REGION Network 11: Е | Ж | З | И | Й |
   RUNG wire#powerrail
      I_Contact( #DONE )
      { S7_Templates := "SrcType := WChar" } EQ_Contact(in1 := #UNICODE, in2 := WCHAR#'Е')
      Move(in := 16#C5, out1 => #ASCII_HEX)
      S_Coil( #DONE )
   END_RUNG
   RUNG wire#powerrail
      I_Contact( #DONE )
      { S7_Templates := "SrcType := WChar" } EQ_Contact(in1 := #UNICODE, in2 := WCHAR#'Ж')
      Move(in := 16#C6, out1 => #ASCII_HEX)
      S_Coil( #DONE )
   END_RUNG
   RUNG wire#powerrail
      I_Contact( #DONE )
      { S7_Templates := "SrcType := WChar" } EQ_Contact(in1 := #UNICODE, in2 := WCHAR#'З')
      Move(in := 16#C7, out1 => #ASCII_HEX)
      S_Coil( #DONE )
   END_RUNG
   RUNG wire#powerrail
      I_Contact( #DONE )
      { S7_Templates := "SrcType := WChar" } EQ_Contact(in1 := #UNICODE, in2 := WCHAR#'И')
      Move(in := 16#C8, out1 => #ASCII_HEX)
      S_Coil( #DONE )
   END_RUNG
   RUNG wire#powerrail
      I_Contact( #DONE )
      { S7_Templates := "SrcType := WChar" } EQ_Contact(in1 := #UNICODE, in2 := WCHAR#'Й')
      Move(in := 16#C9, out1 => #ASCII_HEX)
      S_Coil( #DONE )
   END_RUNG
   // the same network as SCL:
   IF NOT #DONE AND (#UNICODE = WCHAR#'Е') THEN
       #ASCII_HEX := 16#C5;
       #DONE := TRUE;
   END_IF;
   IF NOT #DONE AND (#UNICODE = WCHAR#'Ж') THEN
       #ASCII_HEX := 16#C6;
       #DONE := TRUE;
   END_IF;
   IF NOT #DONE AND (#UNICODE = WCHAR#'З') THEN
       #ASCII_HEX := 16#C7;
       #DONE := TRUE;
   END_IF;
   IF NOT #DONE AND (#UNICODE = WCHAR#'И') THEN
       #ASCII_HEX := 16#C8;
       #DONE := TRUE;
   END_IF;
   IF NOT #DONE AND (#UNICODE = WCHAR#'Й') THEN
       #ASCII_HEX := 16#C9;
       #DONE := TRUE;
   END_IF;
END_REGION

REGION Network 12: К | Л | М | Н | О |
   RUNG wire#powerrail
      I_Contact( #DONE )
      { S7_Templates := "SrcType := WChar" } EQ_Contact(in1 := #UNICODE, in2 := WCHAR#'К')
      Move(in := 16#CA, out1 => #ASCII_HEX)
      S_Coil( #DONE )
   END_RUNG
   RUNG wire#powerrail
      I_Contact( #DONE )
      { S7_Templates := "SrcType := WChar" } EQ_Contact(in1 := #UNICODE, in2 := WCHAR#'Л')
      Move(in := 16#CB, out1 => #ASCII_HEX)
      S_Coil( #DONE )
   END_RUNG
   RUNG wire#powerrail
      I_Contact( #DONE )
      { S7_Templates := "SrcType := WChar" } EQ_Contact(in1 := #UNICODE, in2 := WCHAR#'М')
      Move(in := 16#CC, out1 => #ASCII_HEX)
      S_Coil( #DONE )
   END_RUNG
   RUNG wire#powerrail
      I_Contact( #DONE )
      { S7_Templates := "SrcType := WChar" } EQ_Contact(in1 := #UNICODE, in2 := WCHAR#'Н')
      Move(in := 16#CD, out1 => #ASCII_HEX)
      S_Coil( #DONE )
   END_RUNG
   RUNG wire#powerrail
      I_Contact( #DONE )
      { S7_Templates := "SrcType := WChar" } EQ_Contact(in1 := #UNICODE, in2 := WCHAR#'О')
      Move(in := 16#CE, out1 => #ASCII_HEX)
      S_Coil( #DONE )
   END_RUNG
   // the same network as SCL:
   IF NOT #DONE AND (#UNICODE = WCHAR#'К') THEN
       #ASCII_HEX := 16#CA;
       #DONE := TRUE;
   END_IF;
   IF NOT #DONE AND (#UNICODE = WCHAR#'Л') THEN
       #ASCII_HEX := 16#CB;
       #DONE := TRUE;
   END_IF;
   IF NOT #DONE AND (#UNICODE = WCHAR#'М') THEN
       #ASCII_HEX := 16#CC;
       #DONE := TRUE;
   END_IF;
   IF NOT #DONE AND (#UNICODE = WCHAR#'Н') THEN
       #ASCII_HEX := 16#CD;
       #DONE := TRUE;
   END_IF;
   IF NOT #DONE AND (#UNICODE = WCHAR#'О') THEN
       #ASCII_HEX := 16#CE;
       #DONE := TRUE;
   END_IF;
END_REGION

REGION Network 13: П | Р | С | Т | У |
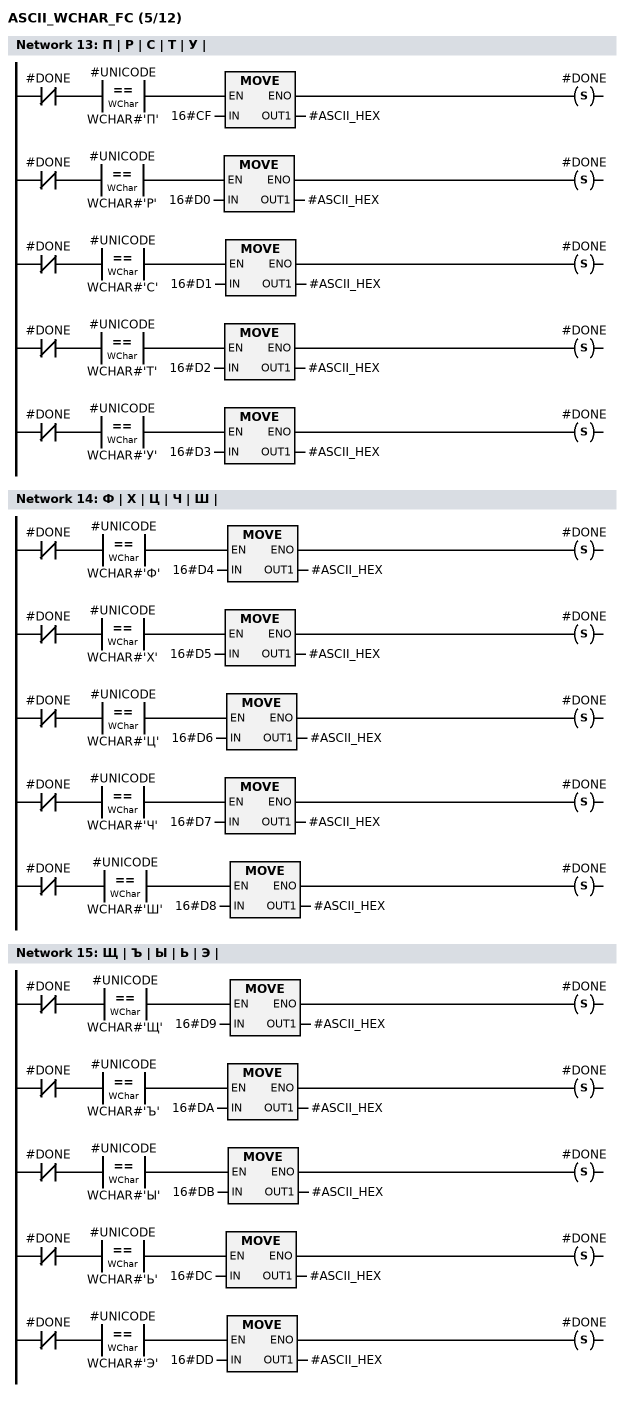
   RUNG wire#powerrail
      I_Contact( #DONE )
      { S7_Templates := "SrcType := WChar" } EQ_Contact(in1 := #UNICODE, in2 := WCHAR#'П')
      Move(in := 16#CF, out1 => #ASCII_HEX)
      S_Coil( #DONE )
   END_RUNG
   RUNG wire#powerrail
      I_Contact( #DONE )
      { S7_Templates := "SrcType := WChar" } EQ_Contact(in1 := #UNICODE, in2 := WCHAR#'Р')
      Move(in := 16#D0, out1 => #ASCII_HEX)
      S_Coil( #DONE )
   END_RUNG
   RUNG wire#powerrail
      I_Contact( #DONE )
      { S7_Templates := "SrcType := WChar" } EQ_Contact(in1 := #UNICODE, in2 := WCHAR#'С')
      Move(in := 16#D1, out1 => #ASCII_HEX)
      S_Coil( #DONE )
   END_RUNG
   RUNG wire#powerrail
      I_Contact( #DONE )
      { S7_Templates := "SrcType := WChar" } EQ_Contact(in1 := #UNICODE, in2 := WCHAR#'Т')
      Move(in := 16#D2, out1 => #ASCII_HEX)
      S_Coil( #DONE )
   END_RUNG
   RUNG wire#powerrail
      I_Contact( #DONE )
      { S7_Templates := "SrcType := WChar" } EQ_Contact(in1 := #UNICODE, in2 := WCHAR#'У')
      Move(in := 16#D3, out1 => #ASCII_HEX)
      S_Coil( #DONE )
   END_RUNG
   // the same network as SCL:
   IF NOT #DONE AND (#UNICODE = WCHAR#'П') THEN
       #ASCII_HEX := 16#CF;
       #DONE := TRUE;
   END_IF;
   IF NOT #DONE AND (#UNICODE = WCHAR#'Р') THEN
       #ASCII_HEX := 16#D0;
       #DONE := TRUE;
   END_IF;
   IF NOT #DONE AND (#UNICODE = WCHAR#'С') THEN
       #ASCII_HEX := 16#D1;
       #DONE := TRUE;
   END_IF;
   IF NOT #DONE AND (#UNICODE = WCHAR#'Т') THEN
       #ASCII_HEX := 16#D2;
       #DONE := TRUE;
   END_IF;
   IF NOT #DONE AND (#UNICODE = WCHAR#'У') THEN
       #ASCII_HEX := 16#D3;
       #DONE := TRUE;
   END_IF;
END_REGION

REGION Network 14: Ф | Х | Ц | Ч | Ш |
   RUNG wire#powerrail
      I_Contact( #DONE )
      { S7_Templates := "SrcType := WChar" } EQ_Contact(in1 := #UNICODE, in2 := WCHAR#'Ф')
      Move(in := 16#D4, out1 => #ASCII_HEX)
      S_Coil( #DONE )
   END_RUNG
   RUNG wire#powerrail
      I_Contact( #DONE )
      { S7_Templates := "SrcType := WChar" } EQ_Contact(in1 := #UNICODE, in2 := WCHAR#'Х')
      Move(in := 16#D5, out1 => #ASCII_HEX)
      S_Coil( #DONE )
   END_RUNG
   RUNG wire#powerrail
      I_Contact( #DONE )
      { S7_Templates := "SrcType := WChar" } EQ_Contact(in1 := #UNICODE, in2 := WCHAR#'Ц')
      Move(in := 16#D6, out1 => #ASCII_HEX)
      S_Coil( #DONE )
   END_RUNG
   RUNG wire#powerrail
      I_Contact( #DONE )
      { S7_Templates := "SrcType := WChar" } EQ_Contact(in1 := #UNICODE, in2 := WCHAR#'Ч')
      Move(in := 16#D7, out1 => #ASCII_HEX)
      S_Coil( #DONE )
   END_RUNG
   RUNG wire#powerrail
      I_Contact( #DONE )
      { S7_Templates := "SrcType := WChar" } EQ_Contact(in1 := #UNICODE, in2 := WCHAR#'Ш')
      Move(in := 16#D8, out1 => #ASCII_HEX)
      S_Coil( #DONE )
   END_RUNG
   // the same network as SCL:
   IF NOT #DONE AND (#UNICODE = WCHAR#'Ф') THEN
       #ASCII_HEX := 16#D4;
       #DONE := TRUE;
   END_IF;
   IF NOT #DONE AND (#UNICODE = WCHAR#'Х') THEN
       #ASCII_HEX := 16#D5;
       #DONE := TRUE;
   END_IF;
   IF NOT #DONE AND (#UNICODE = WCHAR#'Ц') THEN
       #ASCII_HEX := 16#D6;
       #DONE := TRUE;
   END_IF;
   IF NOT #DONE AND (#UNICODE = WCHAR#'Ч') THEN
       #ASCII_HEX := 16#D7;
       #DONE := TRUE;
   END_IF;
   IF NOT #DONE AND (#UNICODE = WCHAR#'Ш') THEN
       #ASCII_HEX := 16#D8;
       #DONE := TRUE;
   END_IF;
END_REGION

REGION Network 15: Щ | Ъ | Ы | Ь | Э |
   RUNG wire#powerrail
      I_Contact( #DONE )
      { S7_Templates := "SrcType := WChar" } EQ_Contact(in1 := #UNICODE, in2 := WCHAR#'Щ')
      Move(in := 16#D9, out1 => #ASCII_HEX)
      S_Coil( #DONE )
   END_RUNG
   RUNG wire#powerrail
      I_Contact( #DONE )
      { S7_Templates := "SrcType := WChar" } EQ_Contact(in1 := #UNICODE, in2 := WCHAR#'Ъ')
      Move(in := 16#DA, out1 => #ASCII_HEX)
      S_Coil( #DONE )
   END_RUNG
   RUNG wire#powerrail
      I_Contact( #DONE )
      { S7_Templates := "SrcType := WChar" } EQ_Contact(in1 := #UNICODE, in2 := WCHAR#'Ы')
      Move(in := 16#DB, out1 => #ASCII_HEX)
      S_Coil( #DONE )
   END_RUNG
   RUNG wire#powerrail
      I_Contact( #DONE )
      { S7_Templates := "SrcType := WChar" } EQ_Contact(in1 := #UNICODE, in2 := WCHAR#'Ь')
      Move(in := 16#DC, out1 => #ASCII_HEX)
      S_Coil( #DONE )
   END_RUNG
   RUNG wire#powerrail
      I_Contact( #DONE )
      { S7_Templates := "SrcType := WChar" } EQ_Contact(in1 := #UNICODE, in2 := WCHAR#'Э')
      Move(in := 16#DD, out1 => #ASCII_HEX)
      S_Coil( #DONE )
   END_RUNG
   // the same network as SCL:
   IF NOT #DONE AND (#UNICODE = WCHAR#'Щ') THEN
       #ASCII_HEX := 16#D9;
       #DONE := TRUE;
   END_IF;
   IF NOT #DONE AND (#UNICODE = WCHAR#'Ъ') THEN
       #ASCII_HEX := 16#DA;
       #DONE := TRUE;
   END_IF;
   IF NOT #DONE AND (#UNICODE = WCHAR#'Ы') THEN
       #ASCII_HEX := 16#DB;
       #DONE := TRUE;
   END_IF;
   IF NOT #DONE AND (#UNICODE = WCHAR#'Ь') THEN
       #ASCII_HEX := 16#DC;
       #DONE := TRUE;
   END_IF;
   IF NOT #DONE AND (#UNICODE = WCHAR#'Э') THEN
       #ASCII_HEX := 16#DD;
       #DONE := TRUE;
   END_IF;
END_REGION

REGION Network 16: Ю | Я |
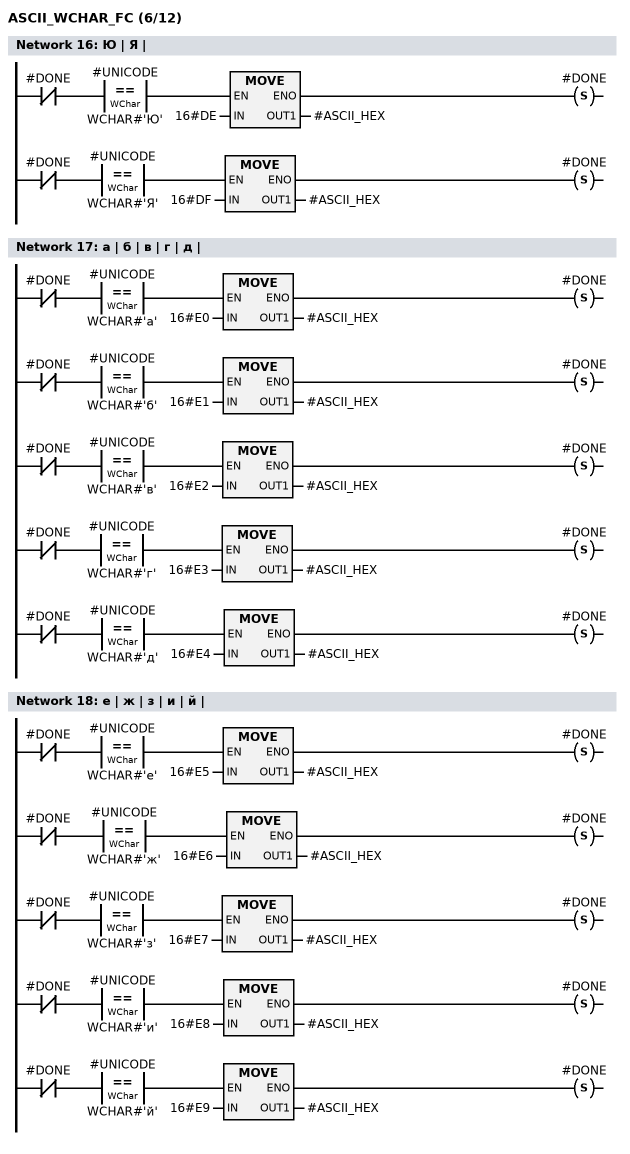
   RUNG wire#powerrail
      I_Contact( #DONE )
      { S7_Templates := "SrcType := WChar" } EQ_Contact(in1 := #UNICODE, in2 := WCHAR#'Ю')
      Move(in := 16#DE, out1 => #ASCII_HEX)
      S_Coil( #DONE )
   END_RUNG
   RUNG wire#powerrail
      I_Contact( #DONE )
      { S7_Templates := "SrcType := WChar" } EQ_Contact(in1 := #UNICODE, in2 := WCHAR#'Я')
      Move(in := 16#DF, out1 => #ASCII_HEX)
      S_Coil( #DONE )
   END_RUNG
   // the same network as SCL:
   IF NOT #DONE AND (#UNICODE = WCHAR#'Ю') THEN
       #ASCII_HEX := 16#DE;
       #DONE := TRUE;
   END_IF;
   IF NOT #DONE AND (#UNICODE = WCHAR#'Я') THEN
       #ASCII_HEX := 16#DF;
       #DONE := TRUE;
   END_IF;
END_REGION

REGION Network 17: а | б | в | г | д |
   RUNG wire#powerrail
      I_Contact( #DONE )
      { S7_Templates := "SrcType := WChar" } EQ_Contact(in1 := #UNICODE, in2 := WCHAR#'а')
      Move(in := 16#E0, out1 => #ASCII_HEX)
      S_Coil( #DONE )
   END_RUNG
   RUNG wire#powerrail
      I_Contact( #DONE )
      { S7_Templates := "SrcType := WChar" } EQ_Contact(in1 := #UNICODE, in2 := WCHAR#'б')
      Move(in := 16#E1, out1 => #ASCII_HEX)
      S_Coil( #DONE )
   END_RUNG
   RUNG wire#powerrail
      I_Contact( #DONE )
      { S7_Templates := "SrcType := WChar" } EQ_Contact(in1 := #UNICODE, in2 := WCHAR#'в')
      Move(in := 16#E2, out1 => #ASCII_HEX)
      S_Coil( #DONE )
   END_RUNG
   RUNG wire#powerrail
      I_Contact( #DONE )
      { S7_Templates := "SrcType := WChar" } EQ_Contact(in1 := #UNICODE, in2 := WCHAR#'г')
      Move(in := 16#E3, out1 => #ASCII_HEX)
      S_Coil( #DONE )
   END_RUNG
   RUNG wire#powerrail
      I_Contact( #DONE )
      { S7_Templates := "SrcType := WChar" } EQ_Contact(in1 := #UNICODE, in2 := WCHAR#'д')
      Move(in := 16#E4, out1 => #ASCII_HEX)
      S_Coil( #DONE )
   END_RUNG
   // the same network as SCL:
   IF NOT #DONE AND (#UNICODE = WCHAR#'а') THEN
       #ASCII_HEX := 16#E0;
       #DONE := TRUE;
   END_IF;
   IF NOT #DONE AND (#UNICODE = WCHAR#'б') THEN
       #ASCII_HEX := 16#E1;
       #DONE := TRUE;
   END_IF;
   IF NOT #DONE AND (#UNICODE = WCHAR#'в') THEN
       #ASCII_HEX := 16#E2;
       #DONE := TRUE;
   END_IF;
   IF NOT #DONE AND (#UNICODE = WCHAR#'г') THEN
       #ASCII_HEX := 16#E3;
       #DONE := TRUE;
   END_IF;
   IF NOT #DONE AND (#UNICODE = WCHAR#'д') THEN
       #ASCII_HEX := 16#E4;
       #DONE := TRUE;
   END_IF;
END_REGION

REGION Network 18: е | ж | з | и | й |
   RUNG wire#powerrail
      I_Contact( #DONE )
      { S7_Templates := "SrcType := WChar" } EQ_Contact(in1 := #UNICODE, in2 := WCHAR#'е')
      Move(in := 16#E5, out1 => #ASCII_HEX)
      S_Coil( #DONE )
   END_RUNG
   RUNG wire#powerrail
      I_Contact( #DONE )
      { S7_Templates := "SrcType := WChar" } EQ_Contact(in1 := #UNICODE, in2 := WCHAR#'ж')
      Move(in := 16#E6, out1 => #ASCII_HEX)
      S_Coil( #DONE )
   END_RUNG
   RUNG wire#powerrail
      I_Contact( #DONE )
      { S7_Templates := "SrcType := WChar" } EQ_Contact(in1 := #UNICODE, in2 := WCHAR#'з')
      Move(in := 16#E7, out1 => #ASCII_HEX)
      S_Coil( #DONE )
   END_RUNG
   RUNG wire#powerrail
      I_Contact( #DONE )
      { S7_Templates := "SrcType := WChar" } EQ_Contact(in1 := #UNICODE, in2 := WCHAR#'и')
      Move(in := 16#E8, out1 => #ASCII_HEX)
      S_Coil( #DONE )
   END_RUNG
   RUNG wire#powerrail
      I_Contact( #DONE )
      { S7_Templates := "SrcType := WChar" } EQ_Contact(in1 := #UNICODE, in2 := WCHAR#'й')
      Move(in := 16#E9, out1 => #ASCII_HEX)
      S_Coil( #DONE )
   END_RUNG
   // the same network as SCL:
   IF NOT #DONE AND (#UNICODE = WCHAR#'е') THEN
       #ASCII_HEX := 16#E5;
       #DONE := TRUE;
   END_IF;
   IF NOT #DONE AND (#UNICODE = WCHAR#'ж') THEN
       #ASCII_HEX := 16#E6;
       #DONE := TRUE;
   END_IF;
   IF NOT #DONE AND (#UNICODE = WCHAR#'з') THEN
       #ASCII_HEX := 16#E7;
       #DONE := TRUE;
   END_IF;
   IF NOT #DONE AND (#UNICODE = WCHAR#'и') THEN
       #ASCII_HEX := 16#E8;
       #DONE := TRUE;
   END_IF;
   IF NOT #DONE AND (#UNICODE = WCHAR#'й') THEN
       #ASCII_HEX := 16#E9;
       #DONE := TRUE;
   END_IF;
END_REGION

REGION Network 19: к | л | м | н | о |
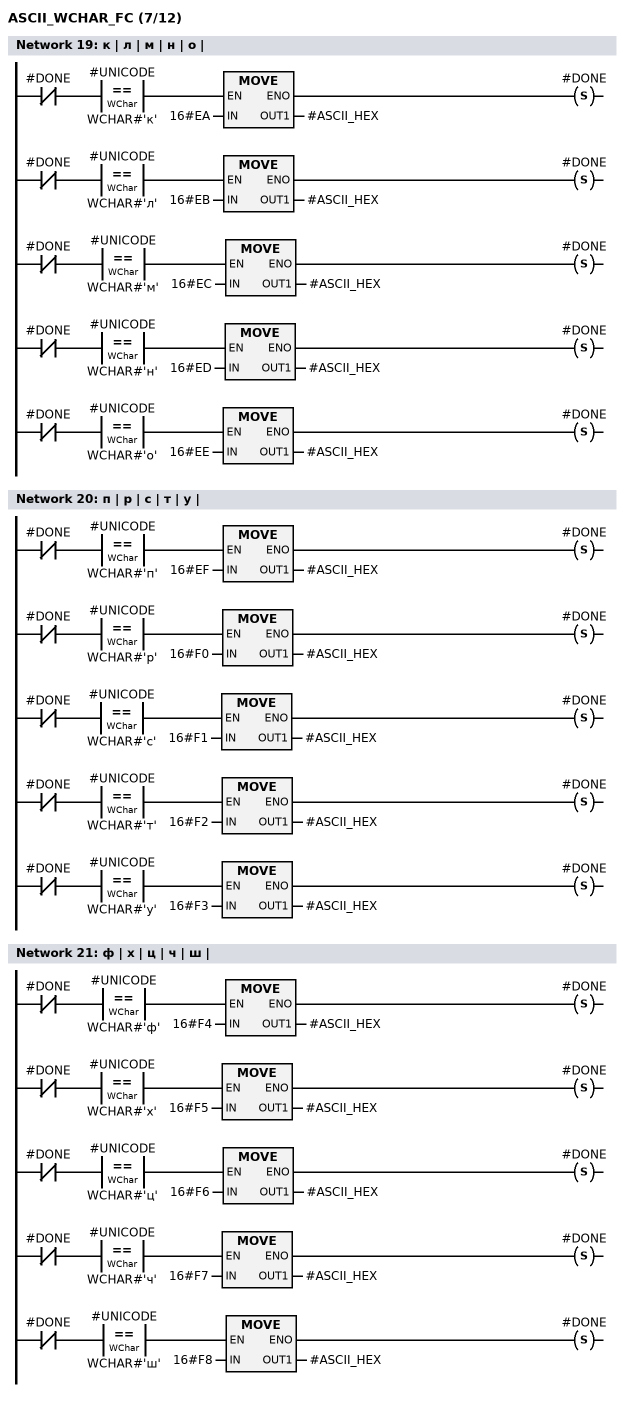
   RUNG wire#powerrail
      I_Contact( #DONE )
      { S7_Templates := "SrcType := WChar" } EQ_Contact(in1 := #UNICODE, in2 := WCHAR#'к')
      Move(in := 16#EA, out1 => #ASCII_HEX)
      S_Coil( #DONE )
   END_RUNG
   RUNG wire#powerrail
      I_Contact( #DONE )
      { S7_Templates := "SrcType := WChar" } EQ_Contact(in1 := #UNICODE, in2 := WCHAR#'л')
      Move(in := 16#EB, out1 => #ASCII_HEX)
      S_Coil( #DONE )
   END_RUNG
   RUNG wire#powerrail
      I_Contact( #DONE )
      { S7_Templates := "SrcType := WChar" } EQ_Contact(in1 := #UNICODE, in2 := WCHAR#'м')
      Move(in := 16#EC, out1 => #ASCII_HEX)
      S_Coil( #DONE )
   END_RUNG
   RUNG wire#powerrail
      I_Contact( #DONE )
      { S7_Templates := "SrcType := WChar" } EQ_Contact(in1 := #UNICODE, in2 := WCHAR#'н')
      Move(in := 16#ED, out1 => #ASCII_HEX)
      S_Coil( #DONE )
   END_RUNG
   RUNG wire#powerrail
      I_Contact( #DONE )
      { S7_Templates := "SrcType := WChar" } EQ_Contact(in1 := #UNICODE, in2 := WCHAR#'о')
      Move(in := 16#EE, out1 => #ASCII_HEX)
      S_Coil( #DONE )
   END_RUNG
   // the same network as SCL:
   IF NOT #DONE AND (#UNICODE = WCHAR#'к') THEN
       #ASCII_HEX := 16#EA;
       #DONE := TRUE;
   END_IF;
   IF NOT #DONE AND (#UNICODE = WCHAR#'л') THEN
       #ASCII_HEX := 16#EB;
       #DONE := TRUE;
   END_IF;
   IF NOT #DONE AND (#UNICODE = WCHAR#'м') THEN
       #ASCII_HEX := 16#EC;
       #DONE := TRUE;
   END_IF;
   IF NOT #DONE AND (#UNICODE = WCHAR#'н') THEN
       #ASCII_HEX := 16#ED;
       #DONE := TRUE;
   END_IF;
   IF NOT #DONE AND (#UNICODE = WCHAR#'о') THEN
       #ASCII_HEX := 16#EE;
       #DONE := TRUE;
   END_IF;
END_REGION

REGION Network 20: п | р | с | т | у |
   RUNG wire#powerrail
      I_Contact( #DONE )
      { S7_Templates := "SrcType := WChar" } EQ_Contact(in1 := #UNICODE, in2 := WCHAR#'п')
      Move(in := 16#EF, out1 => #ASCII_HEX)
      S_Coil( #DONE )
   END_RUNG
   RUNG wire#powerrail
      I_Contact( #DONE )
      { S7_Templates := "SrcType := WChar" } EQ_Contact(in1 := #UNICODE, in2 := WCHAR#'р')
      Move(in := 16#F0, out1 => #ASCII_HEX)
      S_Coil( #DONE )
   END_RUNG
   RUNG wire#powerrail
      I_Contact( #DONE )
      { S7_Templates := "SrcType := WChar" } EQ_Contact(in1 := #UNICODE, in2 := WCHAR#'с')
      Move(in := 16#F1, out1 => #ASCII_HEX)
      S_Coil( #DONE )
   END_RUNG
   RUNG wire#powerrail
      I_Contact( #DONE )
      { S7_Templates := "SrcType := WChar" } EQ_Contact(in1 := #UNICODE, in2 := WCHAR#'т')
      Move(in := 16#F2, out1 => #ASCII_HEX)
      S_Coil( #DONE )
   END_RUNG
   RUNG wire#powerrail
      I_Contact( #DONE )
      { S7_Templates := "SrcType := WChar" } EQ_Contact(in1 := #UNICODE, in2 := WCHAR#'у')
      Move(in := 16#F3, out1 => #ASCII_HEX)
      S_Coil( #DONE )
   END_RUNG
   // the same network as SCL:
   IF NOT #DONE AND (#UNICODE = WCHAR#'п') THEN
       #ASCII_HEX := 16#EF;
       #DONE := TRUE;
   END_IF;
   IF NOT #DONE AND (#UNICODE = WCHAR#'р') THEN
       #ASCII_HEX := 16#F0;
       #DONE := TRUE;
   END_IF;
   IF NOT #DONE AND (#UNICODE = WCHAR#'с') THEN
       #ASCII_HEX := 16#F1;
       #DONE := TRUE;
   END_IF;
   IF NOT #DONE AND (#UNICODE = WCHAR#'т') THEN
       #ASCII_HEX := 16#F2;
       #DONE := TRUE;
   END_IF;
   IF NOT #DONE AND (#UNICODE = WCHAR#'у') THEN
       #ASCII_HEX := 16#F3;
       #DONE := TRUE;
   END_IF;
END_REGION

REGION Network 21: ф | х | ц | ч | ш |
   RUNG wire#powerrail
      I_Contact( #DONE )
      { S7_Templates := "SrcType := WChar" } EQ_Contact(in1 := #UNICODE, in2 := WCHAR#'ф')
      Move(in := 16#F4, out1 => #ASCII_HEX)
      S_Coil( #DONE )
   END_RUNG
   RUNG wire#powerrail
      I_Contact( #DONE )
      { S7_Templates := "SrcType := WChar" } EQ_Contact(in1 := #UNICODE, in2 := WCHAR#'х')
      Move(in := 16#F5, out1 => #ASCII_HEX)
      S_Coil( #DONE )
   END_RUNG
   RUNG wire#powerrail
      I_Contact( #DONE )
      { S7_Templates := "SrcType := WChar" } EQ_Contact(in1 := #UNICODE, in2 := WCHAR#'ц')
      Move(in := 16#F6, out1 => #ASCII_HEX)
      S_Coil( #DONE )
   END_RUNG
   RUNG wire#powerrail
      I_Contact( #DONE )
      { S7_Templates := "SrcType := WChar" } EQ_Contact(in1 := #UNICODE, in2 := WCHAR#'ч')
      Move(in := 16#F7, out1 => #ASCII_HEX)
      S_Coil( #DONE )
   END_RUNG
   RUNG wire#powerrail
      I_Contact( #DONE )
      { S7_Templates := "SrcType := WChar" } EQ_Contact(in1 := #UNICODE, in2 := WCHAR#'ш')
      Move(in := 16#F8, out1 => #ASCII_HEX)
      S_Coil( #DONE )
   END_RUNG
   // the same network as SCL:
   IF NOT #DONE AND (#UNICODE = WCHAR#'ф') THEN
       #ASCII_HEX := 16#F4;
       #DONE := TRUE;
   END_IF;
   IF NOT #DONE AND (#UNICODE = WCHAR#'х') THEN
       #ASCII_HEX := 16#F5;
       #DONE := TRUE;
   END_IF;
   IF NOT #DONE AND (#UNICODE = WCHAR#'ц') THEN
       #ASCII_HEX := 16#F6;
       #DONE := TRUE;
   END_IF;
   IF NOT #DONE AND (#UNICODE = WCHAR#'ч') THEN
       #ASCII_HEX := 16#F7;
       #DONE := TRUE;
   END_IF;
   IF NOT #DONE AND (#UNICODE = WCHAR#'ш') THEN
       #ASCII_HEX := 16#F8;
       #DONE := TRUE;
   END_IF;
END_REGION

REGION Network 22: щ | ъ | ы | ь | э |
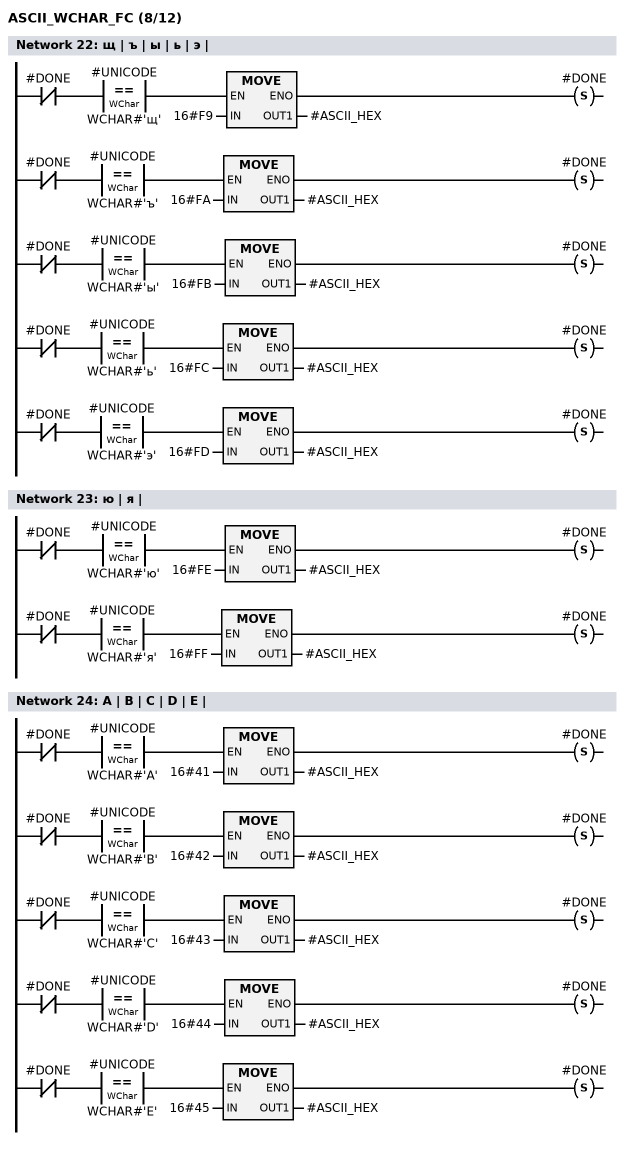
   RUNG wire#powerrail
      I_Contact( #DONE )
      { S7_Templates := "SrcType := WChar" } EQ_Contact(in1 := #UNICODE, in2 := WCHAR#'щ')
      Move(in := 16#F9, out1 => #ASCII_HEX)
      S_Coil( #DONE )
   END_RUNG
   RUNG wire#powerrail
      I_Contact( #DONE )
      { S7_Templates := "SrcType := WChar" } EQ_Contact(in1 := #UNICODE, in2 := WCHAR#'ъ')
      Move(in := 16#FA, out1 => #ASCII_HEX)
      S_Coil( #DONE )
   END_RUNG
   RUNG wire#powerrail
      I_Contact( #DONE )
      { S7_Templates := "SrcType := WChar" } EQ_Contact(in1 := #UNICODE, in2 := WCHAR#'ы')
      Move(in := 16#FB, out1 => #ASCII_HEX)
      S_Coil( #DONE )
   END_RUNG
   RUNG wire#powerrail
      I_Contact( #DONE )
      { S7_Templates := "SrcType := WChar" } EQ_Contact(in1 := #UNICODE, in2 := WCHAR#'ь')
      Move(in := 16#FC, out1 => #ASCII_HEX)
      S_Coil( #DONE )
   END_RUNG
   RUNG wire#powerrail
      I_Contact( #DONE )
      { S7_Templates := "SrcType := WChar" } EQ_Contact(in1 := #UNICODE, in2 := WCHAR#'э')
      Move(in := 16#FD, out1 => #ASCII_HEX)
      S_Coil( #DONE )
   END_RUNG
   // the same network as SCL:
   IF NOT #DONE AND (#UNICODE = WCHAR#'щ') THEN
       #ASCII_HEX := 16#F9;
       #DONE := TRUE;
   END_IF;
   IF NOT #DONE AND (#UNICODE = WCHAR#'ъ') THEN
       #ASCII_HEX := 16#FA;
       #DONE := TRUE;
   END_IF;
   IF NOT #DONE AND (#UNICODE = WCHAR#'ы') THEN
       #ASCII_HEX := 16#FB;
       #DONE := TRUE;
   END_IF;
   IF NOT #DONE AND (#UNICODE = WCHAR#'ь') THEN
       #ASCII_HEX := 16#FC;
       #DONE := TRUE;
   END_IF;
   IF NOT #DONE AND (#UNICODE = WCHAR#'э') THEN
       #ASCII_HEX := 16#FD;
       #DONE := TRUE;
   END_IF;
END_REGION

REGION Network 23: ю | я |
   RUNG wire#powerrail
      I_Contact( #DONE )
      { S7_Templates := "SrcType := WChar" } EQ_Contact(in1 := #UNICODE, in2 := WCHAR#'ю')
      Move(in := 16#FE, out1 => #ASCII_HEX)
      S_Coil( #DONE )
   END_RUNG
   RUNG wire#powerrail
      I_Contact( #DONE )
      { S7_Templates := "SrcType := WChar" } EQ_Contact(in1 := #UNICODE, in2 := WCHAR#'я')
      Move(in := 16#FF, out1 => #ASCII_HEX)
      S_Coil( #DONE )
   END_RUNG
   // the same network as SCL:
   IF NOT #DONE AND (#UNICODE = WCHAR#'ю') THEN
       #ASCII_HEX := 16#FE;
       #DONE := TRUE;
   END_IF;
   IF NOT #DONE AND (#UNICODE = WCHAR#'я') THEN
       #ASCII_HEX := 16#FF;
       #DONE := TRUE;
   END_IF;
END_REGION

REGION Network 24: A | B | C | D | E |
   RUNG wire#powerrail
      I_Contact( #DONE )
      { S7_Templates := "SrcType := WChar" } EQ_Contact(in1 := #UNICODE, in2 := WCHAR#'A')
      Move(in := 16#41, out1 => #ASCII_HEX)
      S_Coil( #DONE )
   END_RUNG
   RUNG wire#powerrail
      I_Contact( #DONE )
      { S7_Templates := "SrcType := WChar" } EQ_Contact(in1 := #UNICODE, in2 := WCHAR#'B')
      Move(in := 16#42, out1 => #ASCII_HEX)
      S_Coil( #DONE )
   END_RUNG
   RUNG wire#powerrail
      I_Contact( #DONE )
      { S7_Templates := "SrcType := WChar" } EQ_Contact(in1 := #UNICODE, in2 := WCHAR#'C')
      Move(in := 16#43, out1 => #ASCII_HEX)
      S_Coil( #DONE )
   END_RUNG
   RUNG wire#powerrail
      I_Contact( #DONE )
      { S7_Templates := "SrcType := WChar" } EQ_Contact(in1 := #UNICODE, in2 := WCHAR#'D')
      Move(in := 16#44, out1 => #ASCII_HEX)
      S_Coil( #DONE )
   END_RUNG
   RUNG wire#powerrail
      I_Contact( #DONE )
      { S7_Templates := "SrcType := WChar" } EQ_Contact(in1 := #UNICODE, in2 := WCHAR#'E')
      Move(in := 16#45, out1 => #ASCII_HEX)
      S_Coil( #DONE )
   END_RUNG
   // the same network as SCL:
   IF NOT #DONE AND (#UNICODE = WCHAR#'A') THEN
       #ASCII_HEX := 16#41;
       #DONE := TRUE;
   END_IF;
   IF NOT #DONE AND (#UNICODE = WCHAR#'B') THEN
       #ASCII_HEX := 16#42;
       #DONE := TRUE;
   END_IF;
   IF NOT #DONE AND (#UNICODE = WCHAR#'C') THEN
       #ASCII_HEX := 16#43;
       #DONE := TRUE;
   END_IF;
   IF NOT #DONE AND (#UNICODE = WCHAR#'D') THEN
       #ASCII_HEX := 16#44;
       #DONE := TRUE;
   END_IF;
   IF NOT #DONE AND (#UNICODE = WCHAR#'E') THEN
       #ASCII_HEX := 16#45;
       #DONE := TRUE;
   END_IF;
END_REGION

REGION Network 25: F | G | H | I | J |
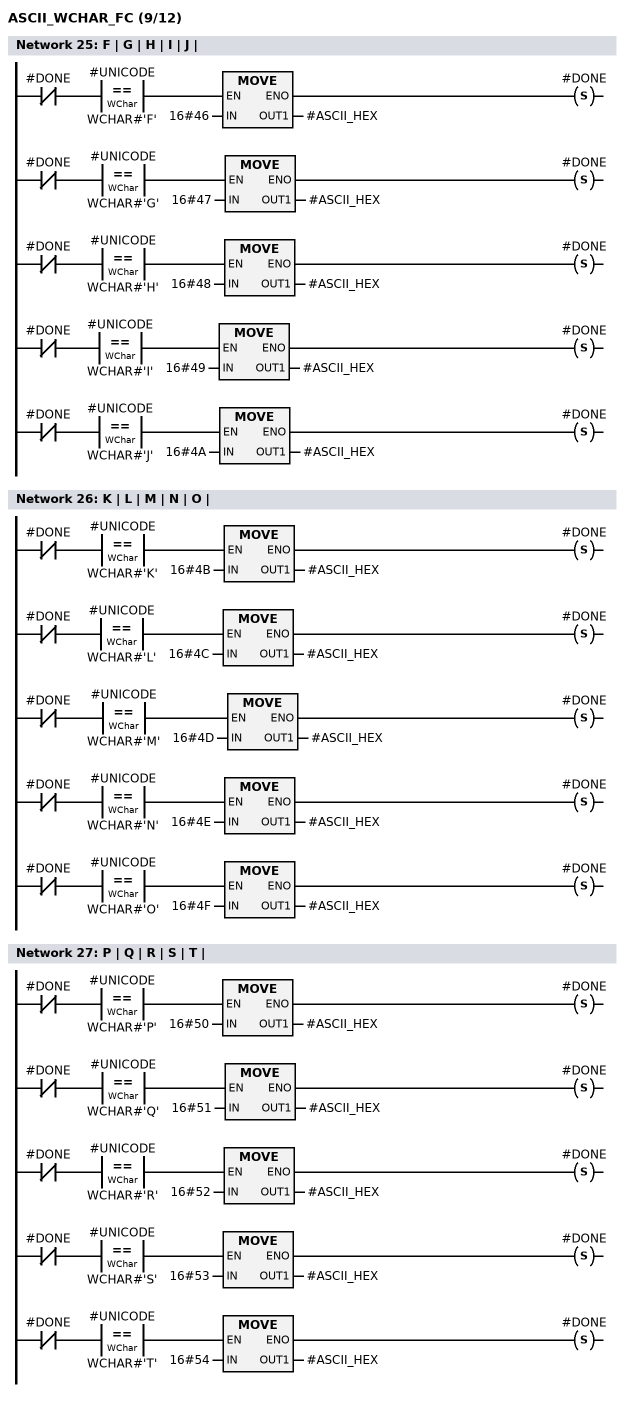
   RUNG wire#powerrail
      I_Contact( #DONE )
      { S7_Templates := "SrcType := WChar" } EQ_Contact(in1 := #UNICODE, in2 := WCHAR#'F')
      Move(in := 16#46, out1 => #ASCII_HEX)
      S_Coil( #DONE )
   END_RUNG
   RUNG wire#powerrail
      I_Contact( #DONE )
      { S7_Templates := "SrcType := WChar" } EQ_Contact(in1 := #UNICODE, in2 := WCHAR#'G')
      Move(in := 16#47, out1 => #ASCII_HEX)
      S_Coil( #DONE )
   END_RUNG
   RUNG wire#powerrail
      I_Contact( #DONE )
      { S7_Templates := "SrcType := WChar" } EQ_Contact(in1 := #UNICODE, in2 := WCHAR#'H')
      Move(in := 16#48, out1 => #ASCII_HEX)
      S_Coil( #DONE )
   END_RUNG
   RUNG wire#powerrail
      I_Contact( #DONE )
      { S7_Templates := "SrcType := WChar" } EQ_Contact(in1 := #UNICODE, in2 := WCHAR#'I')
      Move(in := 16#49, out1 => #ASCII_HEX)
      S_Coil( #DONE )
   END_RUNG
   RUNG wire#powerrail
      I_Contact( #DONE )
      { S7_Templates := "SrcType := WChar" } EQ_Contact(in1 := #UNICODE, in2 := WCHAR#'J')
      Move(in := 16#4A, out1 => #ASCII_HEX)
      S_Coil( #DONE )
   END_RUNG
   // the same network as SCL:
   IF NOT #DONE AND (#UNICODE = WCHAR#'F') THEN
       #ASCII_HEX := 16#46;
       #DONE := TRUE;
   END_IF;
   IF NOT #DONE AND (#UNICODE = WCHAR#'G') THEN
       #ASCII_HEX := 16#47;
       #DONE := TRUE;
   END_IF;
   IF NOT #DONE AND (#UNICODE = WCHAR#'H') THEN
       #ASCII_HEX := 16#48;
       #DONE := TRUE;
   END_IF;
   IF NOT #DONE AND (#UNICODE = WCHAR#'I') THEN
       #ASCII_HEX := 16#49;
       #DONE := TRUE;
   END_IF;
   IF NOT #DONE AND (#UNICODE = WCHAR#'J') THEN
       #ASCII_HEX := 16#4A;
       #DONE := TRUE;
   END_IF;
END_REGION

REGION Network 26: K | L | M | N | O |
   RUNG wire#powerrail
      I_Contact( #DONE )
      { S7_Templates := "SrcType := WChar" } EQ_Contact(in1 := #UNICODE, in2 := WCHAR#'K')
      Move(in := 16#4B, out1 => #ASCII_HEX)
      S_Coil( #DONE )
   END_RUNG
   RUNG wire#powerrail
      I_Contact( #DONE )
      { S7_Templates := "SrcType := WChar" } EQ_Contact(in1 := #UNICODE, in2 := WCHAR#'L')
      Move(in := 16#4C, out1 => #ASCII_HEX)
      S_Coil( #DONE )
   END_RUNG
   RUNG wire#powerrail
      I_Contact( #DONE )
      { S7_Templates := "SrcType := WChar" } EQ_Contact(in1 := #UNICODE, in2 := WCHAR#'M')
      Move(in := 16#4D, out1 => #ASCII_HEX)
      S_Coil( #DONE )
   END_RUNG
   RUNG wire#powerrail
      I_Contact( #DONE )
      { S7_Templates := "SrcType := WChar" } EQ_Contact(in1 := #UNICODE, in2 := WCHAR#'N')
      Move(in := 16#4E, out1 => #ASCII_HEX)
      S_Coil( #DONE )
   END_RUNG
   RUNG wire#powerrail
      I_Contact( #DONE )
      { S7_Templates := "SrcType := WChar" } EQ_Contact(in1 := #UNICODE, in2 := WCHAR#'O')
      Move(in := 16#4F, out1 => #ASCII_HEX)
      S_Coil( #DONE )
   END_RUNG
   // the same network as SCL:
   IF NOT #DONE AND (#UNICODE = WCHAR#'K') THEN
       #ASCII_HEX := 16#4B;
       #DONE := TRUE;
   END_IF;
   IF NOT #DONE AND (#UNICODE = WCHAR#'L') THEN
       #ASCII_HEX := 16#4C;
       #DONE := TRUE;
   END_IF;
   IF NOT #DONE AND (#UNICODE = WCHAR#'M') THEN
       #ASCII_HEX := 16#4D;
       #DONE := TRUE;
   END_IF;
   IF NOT #DONE AND (#UNICODE = WCHAR#'N') THEN
       #ASCII_HEX := 16#4E;
       #DONE := TRUE;
   END_IF;
   IF NOT #DONE AND (#UNICODE = WCHAR#'O') THEN
       #ASCII_HEX := 16#4F;
       #DONE := TRUE;
   END_IF;
END_REGION

REGION Network 27: P | Q | R | S | T |
   RUNG wire#powerrail
      I_Contact( #DONE )
      { S7_Templates := "SrcType := WChar" } EQ_Contact(in1 := #UNICODE, in2 := WCHAR#'P')
      Move(in := 16#50, out1 => #ASCII_HEX)
      S_Coil( #DONE )
   END_RUNG
   RUNG wire#powerrail
      I_Contact( #DONE )
      { S7_Templates := "SrcType := WChar" } EQ_Contact(in1 := #UNICODE, in2 := WCHAR#'Q')
      Move(in := 16#51, out1 => #ASCII_HEX)
      S_Coil( #DONE )
   END_RUNG
   RUNG wire#powerrail
      I_Contact( #DONE )
      { S7_Templates := "SrcType := WChar" } EQ_Contact(in1 := #UNICODE, in2 := WCHAR#'R')
      Move(in := 16#52, out1 => #ASCII_HEX)
      S_Coil( #DONE )
   END_RUNG
   RUNG wire#powerrail
      I_Contact( #DONE )
      { S7_Templates := "SrcType := WChar" } EQ_Contact(in1 := #UNICODE, in2 := WCHAR#'S')
      Move(in := 16#53, out1 => #ASCII_HEX)
      S_Coil( #DONE )
   END_RUNG
   RUNG wire#powerrail
      I_Contact( #DONE )
      { S7_Templates := "SrcType := WChar" } EQ_Contact(in1 := #UNICODE, in2 := WCHAR#'T')
      Move(in := 16#54, out1 => #ASCII_HEX)
      S_Coil( #DONE )
   END_RUNG
   // the same network as SCL:
   IF NOT #DONE AND (#UNICODE = WCHAR#'P') THEN
       #ASCII_HEX := 16#50;
       #DONE := TRUE;
   END_IF;
   IF NOT #DONE AND (#UNICODE = WCHAR#'Q') THEN
       #ASCII_HEX := 16#51;
       #DONE := TRUE;
   END_IF;
   IF NOT #DONE AND (#UNICODE = WCHAR#'R') THEN
       #ASCII_HEX := 16#52;
       #DONE := TRUE;
   END_IF;
   IF NOT #DONE AND (#UNICODE = WCHAR#'S') THEN
       #ASCII_HEX := 16#53;
       #DONE := TRUE;
   END_IF;
   IF NOT #DONE AND (#UNICODE = WCHAR#'T') THEN
       #ASCII_HEX := 16#54;
       #DONE := TRUE;
   END_IF;
END_REGION

REGION Network 28: U | V | W | X | Y | Z |
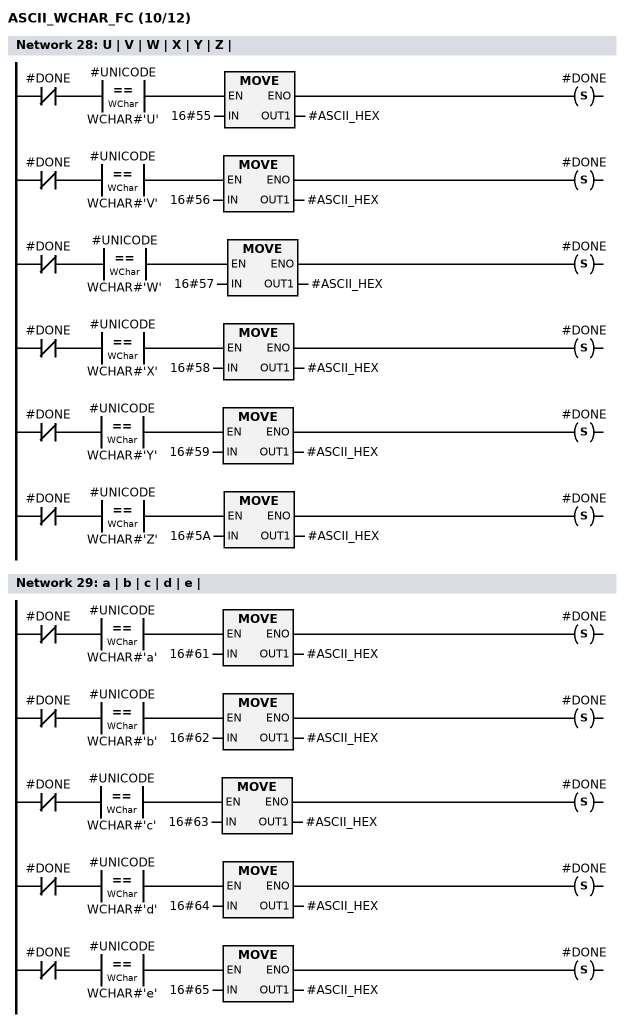
   RUNG wire#powerrail
      I_Contact( #DONE )
      { S7_Templates := "SrcType := WChar" } EQ_Contact(in1 := #UNICODE, in2 := WCHAR#'U')
      Move(in := 16#55, out1 => #ASCII_HEX)
      S_Coil( #DONE )
   END_RUNG
   RUNG wire#powerrail
      I_Contact( #DONE )
      { S7_Templates := "SrcType := WChar" } EQ_Contact(in1 := #UNICODE, in2 := WCHAR#'V')
      Move(in := 16#56, out1 => #ASCII_HEX)
      S_Coil( #DONE )
   END_RUNG
   RUNG wire#powerrail
      I_Contact( #DONE )
      { S7_Templates := "SrcType := WChar" } EQ_Contact(in1 := #UNICODE, in2 := WCHAR#'W')
      Move(in := 16#57, out1 => #ASCII_HEX)
      S_Coil( #DONE )
   END_RUNG
   RUNG wire#powerrail
      I_Contact( #DONE )
      { S7_Templates := "SrcType := WChar" } EQ_Contact(in1 := #UNICODE, in2 := WCHAR#'X')
      Move(in := 16#58, out1 => #ASCII_HEX)
      S_Coil( #DONE )
   END_RUNG
   RUNG wire#powerrail
      I_Contact( #DONE )
      { S7_Templates := "SrcType := WChar" } EQ_Contact(in1 := #UNICODE, in2 := WCHAR#'Y')
      Move(in := 16#59, out1 => #ASCII_HEX)
      S_Coil( #DONE )
   END_RUNG
   RUNG wire#powerrail
      I_Contact( #DONE )
      { S7_Templates := "SrcType := WChar" } EQ_Contact(in1 := #UNICODE, in2 := WCHAR#'Z')
      Move(in := 16#5A, out1 => #ASCII_HEX)
      S_Coil( #DONE )
   END_RUNG
   // the same network as SCL:
   IF NOT #DONE AND (#UNICODE = WCHAR#'U') THEN
       #ASCII_HEX := 16#55;
       #DONE := TRUE;
   END_IF;
   IF NOT #DONE AND (#UNICODE = WCHAR#'V') THEN
       #ASCII_HEX := 16#56;
       #DONE := TRUE;
   END_IF;
   IF NOT #DONE AND (#UNICODE = WCHAR#'W') THEN
       #ASCII_HEX := 16#57;
       #DONE := TRUE;
   END_IF;
   IF NOT #DONE AND (#UNICODE = WCHAR#'X') THEN
       #ASCII_HEX := 16#58;
       #DONE := TRUE;
   END_IF;
   IF NOT #DONE AND (#UNICODE = WCHAR#'Y') THEN
       #ASCII_HEX := 16#59;
       #DONE := TRUE;
   END_IF;
   IF NOT #DONE AND (#UNICODE = WCHAR#'Z') THEN
       #ASCII_HEX := 16#5A;
       #DONE := TRUE;
   END_IF;
END_REGION

REGION Network 29: a | b | c | d | e |
   RUNG wire#powerrail
      I_Contact( #DONE )
      { S7_Templates := "SrcType := WChar" } EQ_Contact(in1 := #UNICODE, in2 := WCHAR#'a')
      Move(in := 16#61, out1 => #ASCII_HEX)
      S_Coil( #DONE )
   END_RUNG
   RUNG wire#powerrail
      I_Contact( #DONE )
      { S7_Templates := "SrcType := WChar" } EQ_Contact(in1 := #UNICODE, in2 := WCHAR#'b')
      Move(in := 16#62, out1 => #ASCII_HEX)
      S_Coil( #DONE )
   END_RUNG
   RUNG wire#powerrail
      I_Contact( #DONE )
      { S7_Templates := "SrcType := WChar" } EQ_Contact(in1 := #UNICODE, in2 := WCHAR#'c')
      Move(in := 16#63, out1 => #ASCII_HEX)
      S_Coil( #DONE )
   END_RUNG
   RUNG wire#powerrail
      I_Contact( #DONE )
      { S7_Templates := "SrcType := WChar" } EQ_Contact(in1 := #UNICODE, in2 := WCHAR#'d')
      Move(in := 16#64, out1 => #ASCII_HEX)
      S_Coil( #DONE )
   END_RUNG
   RUNG wire#powerrail
      I_Contact( #DONE )
      { S7_Templates := "SrcType := WChar" } EQ_Contact(in1 := #UNICODE, in2 := WCHAR#'e')
      Move(in := 16#65, out1 => #ASCII_HEX)
      S_Coil( #DONE )
   END_RUNG
   // the same network as SCL:
   IF NOT #DONE AND (#UNICODE = WCHAR#'a') THEN
       #ASCII_HEX := 16#61;
       #DONE := TRUE;
   END_IF;
   IF NOT #DONE AND (#UNICODE = WCHAR#'b') THEN
       #ASCII_HEX := 16#62;
       #DONE := TRUE;
   END_IF;
   IF NOT #DONE AND (#UNICODE = WCHAR#'c') THEN
       #ASCII_HEX := 16#63;
       #DONE := TRUE;
   END_IF;
   IF NOT #DONE AND (#UNICODE = WCHAR#'d') THEN
       #ASCII_HEX := 16#64;
       #DONE := TRUE;
   END_IF;
   IF NOT #DONE AND (#UNICODE = WCHAR#'e') THEN
       #ASCII_HEX := 16#65;
       #DONE := TRUE;
   END_IF;
END_REGION

REGION Network 30: f | g | h | i | j |
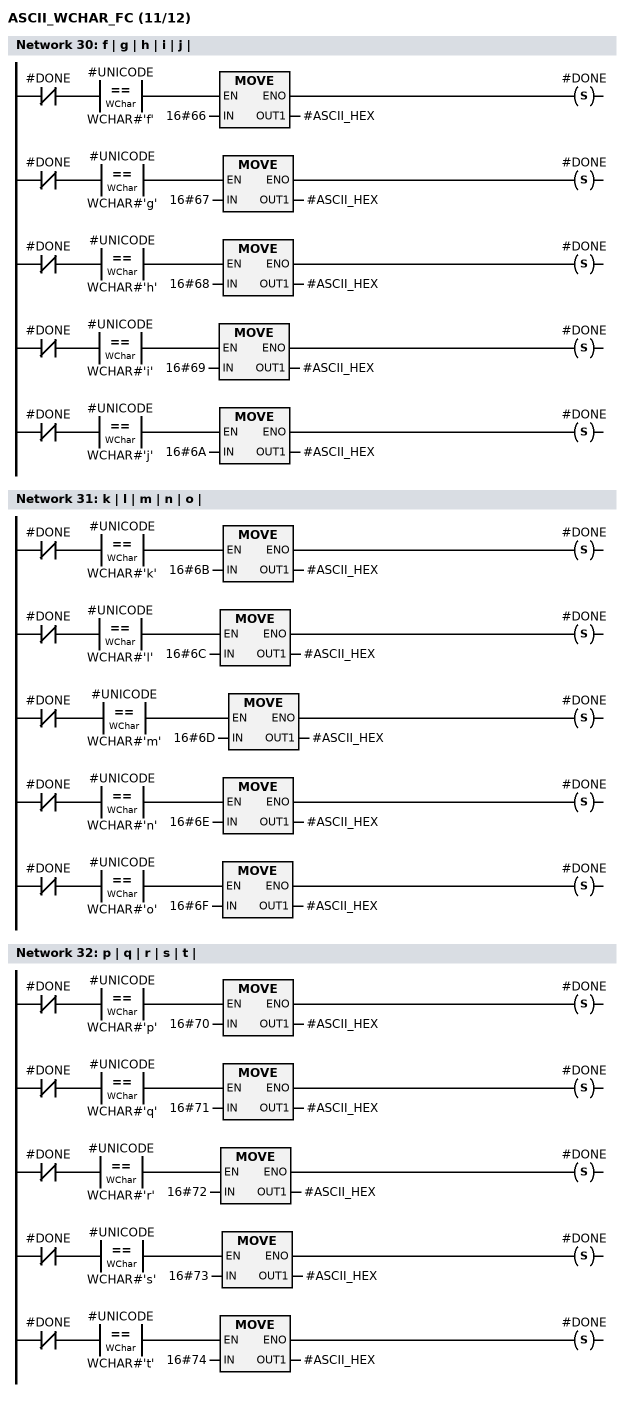
   RUNG wire#powerrail
      I_Contact( #DONE )
      { S7_Templates := "SrcType := WChar" } EQ_Contact(in1 := #UNICODE, in2 := WCHAR#'f')
      Move(in := 16#66, out1 => #ASCII_HEX)
      S_Coil( #DONE )
   END_RUNG
   RUNG wire#powerrail
      I_Contact( #DONE )
      { S7_Templates := "SrcType := WChar" } EQ_Contact(in1 := #UNICODE, in2 := WCHAR#'g')
      Move(in := 16#67, out1 => #ASCII_HEX)
      S_Coil( #DONE )
   END_RUNG
   RUNG wire#powerrail
      I_Contact( #DONE )
      { S7_Templates := "SrcType := WChar" } EQ_Contact(in1 := #UNICODE, in2 := WCHAR#'h')
      Move(in := 16#68, out1 => #ASCII_HEX)
      S_Coil( #DONE )
   END_RUNG
   RUNG wire#powerrail
      I_Contact( #DONE )
      { S7_Templates := "SrcType := WChar" } EQ_Contact(in1 := #UNICODE, in2 := WCHAR#'i')
      Move(in := 16#69, out1 => #ASCII_HEX)
      S_Coil( #DONE )
   END_RUNG
   RUNG wire#powerrail
      I_Contact( #DONE )
      { S7_Templates := "SrcType := WChar" } EQ_Contact(in1 := #UNICODE, in2 := WCHAR#'j')
      Move(in := 16#6A, out1 => #ASCII_HEX)
      S_Coil( #DONE )
   END_RUNG
   // the same network as SCL:
   IF NOT #DONE AND (#UNICODE = WCHAR#'f') THEN
       #ASCII_HEX := 16#66;
       #DONE := TRUE;
   END_IF;
   IF NOT #DONE AND (#UNICODE = WCHAR#'g') THEN
       #ASCII_HEX := 16#67;
       #DONE := TRUE;
   END_IF;
   IF NOT #DONE AND (#UNICODE = WCHAR#'h') THEN
       #ASCII_HEX := 16#68;
       #DONE := TRUE;
   END_IF;
   IF NOT #DONE AND (#UNICODE = WCHAR#'i') THEN
       #ASCII_HEX := 16#69;
       #DONE := TRUE;
   END_IF;
   IF NOT #DONE AND (#UNICODE = WCHAR#'j') THEN
       #ASCII_HEX := 16#6A;
       #DONE := TRUE;
   END_IF;
END_REGION

REGION Network 31: k | l | m | n | o |
   RUNG wire#powerrail
      I_Contact( #DONE )
      { S7_Templates := "SrcType := WChar" } EQ_Contact(in1 := #UNICODE, in2 := WCHAR#'k')
      Move(in := 16#6B, out1 => #ASCII_HEX)
      S_Coil( #DONE )
   END_RUNG
   RUNG wire#powerrail
      I_Contact( #DONE )
      { S7_Templates := "SrcType := WChar" } EQ_Contact(in1 := #UNICODE, in2 := WCHAR#'l')
      Move(in := 16#6C, out1 => #ASCII_HEX)
      S_Coil( #DONE )
   END_RUNG
   RUNG wire#powerrail
      I_Contact( #DONE )
      { S7_Templates := "SrcType := WChar" } EQ_Contact(in1 := #UNICODE, in2 := WCHAR#'m')
      Move(in := 16#6D, out1 => #ASCII_HEX)
      S_Coil( #DONE )
   END_RUNG
   RUNG wire#powerrail
      I_Contact( #DONE )
      { S7_Templates := "SrcType := WChar" } EQ_Contact(in1 := #UNICODE, in2 := WCHAR#'n')
      Move(in := 16#6E, out1 => #ASCII_HEX)
      S_Coil( #DONE )
   END_RUNG
   RUNG wire#powerrail
      I_Contact( #DONE )
      { S7_Templates := "SrcType := WChar" } EQ_Contact(in1 := #UNICODE, in2 := WCHAR#'o')
      Move(in := 16#6F, out1 => #ASCII_HEX)
      S_Coil( #DONE )
   END_RUNG
   // the same network as SCL:
   IF NOT #DONE AND (#UNICODE = WCHAR#'k') THEN
       #ASCII_HEX := 16#6B;
       #DONE := TRUE;
   END_IF;
   IF NOT #DONE AND (#UNICODE = WCHAR#'l') THEN
       #ASCII_HEX := 16#6C;
       #DONE := TRUE;
   END_IF;
   IF NOT #DONE AND (#UNICODE = WCHAR#'m') THEN
       #ASCII_HEX := 16#6D;
       #DONE := TRUE;
   END_IF;
   IF NOT #DONE AND (#UNICODE = WCHAR#'n') THEN
       #ASCII_HEX := 16#6E;
       #DONE := TRUE;
   END_IF;
   IF NOT #DONE AND (#UNICODE = WCHAR#'o') THEN
       #ASCII_HEX := 16#6F;
       #DONE := TRUE;
   END_IF;
END_REGION

REGION Network 32: p | q | r | s | t |
   RUNG wire#powerrail
      I_Contact( #DONE )
      { S7_Templates := "SrcType := WChar" } EQ_Contact(in1 := #UNICODE, in2 := WCHAR#'p')
      Move(in := 16#70, out1 => #ASCII_HEX)
      S_Coil( #DONE )
   END_RUNG
   RUNG wire#powerrail
      I_Contact( #DONE )
      { S7_Templates := "SrcType := WChar" } EQ_Contact(in1 := #UNICODE, in2 := WCHAR#'q')
      Move(in := 16#71, out1 => #ASCII_HEX)
      S_Coil( #DONE )
   END_RUNG
   RUNG wire#powerrail
      I_Contact( #DONE )
      { S7_Templates := "SrcType := WChar" } EQ_Contact(in1 := #UNICODE, in2 := WCHAR#'r')
      Move(in := 16#72, out1 => #ASCII_HEX)
      S_Coil( #DONE )
   END_RUNG
   RUNG wire#powerrail
      I_Contact( #DONE )
      { S7_Templates := "SrcType := WChar" } EQ_Contact(in1 := #UNICODE, in2 := WCHAR#'s')
      Move(in := 16#73, out1 => #ASCII_HEX)
      S_Coil( #DONE )
   END_RUNG
   RUNG wire#powerrail
      I_Contact( #DONE )
      { S7_Templates := "SrcType := WChar" } EQ_Contact(in1 := #UNICODE, in2 := WCHAR#'t')
      Move(in := 16#74, out1 => #ASCII_HEX)
      S_Coil( #DONE )
   END_RUNG
   // the same network as SCL:
   IF NOT #DONE AND (#UNICODE = WCHAR#'p') THEN
       #ASCII_HEX := 16#70;
       #DONE := TRUE;
   END_IF;
   IF NOT #DONE AND (#UNICODE = WCHAR#'q') THEN
       #ASCII_HEX := 16#71;
       #DONE := TRUE;
   END_IF;
   IF NOT #DONE AND (#UNICODE = WCHAR#'r') THEN
       #ASCII_HEX := 16#72;
       #DONE := TRUE;
   END_IF;
   IF NOT #DONE AND (#UNICODE = WCHAR#'s') THEN
       #ASCII_HEX := 16#73;
       #DONE := TRUE;
   END_IF;
   IF NOT #DONE AND (#UNICODE = WCHAR#'t') THEN
       #ASCII_HEX := 16#74;
       #DONE := TRUE;
   END_IF;
END_REGION

REGION Network 33: u | v | w | x | y | z |
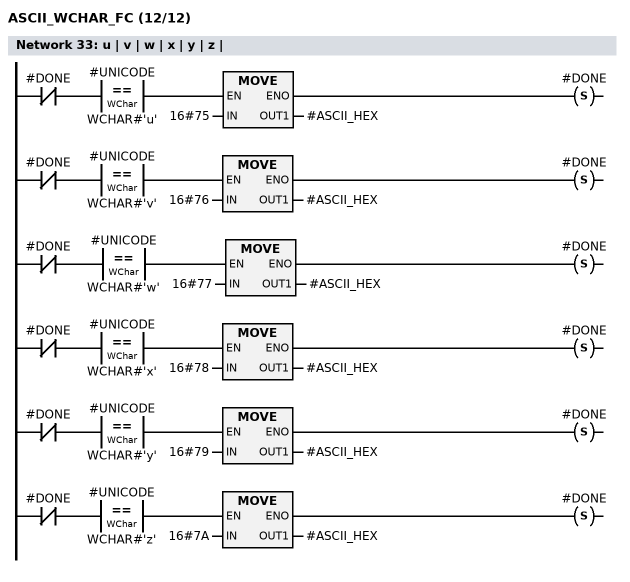
   RUNG wire#powerrail
      I_Contact( #DONE )
      { S7_Templates := "SrcType := WChar" } EQ_Contact(in1 := #UNICODE, in2 := WCHAR#'u')
      Move(in := 16#75, out1 => #ASCII_HEX)
      S_Coil( #DONE )
   END_RUNG
   RUNG wire#powerrail
      I_Contact( #DONE )
      { S7_Templates := "SrcType := WChar" } EQ_Contact(in1 := #UNICODE, in2 := WCHAR#'v')
      Move(in := 16#76, out1 => #ASCII_HEX)
      S_Coil( #DONE )
   END_RUNG
   RUNG wire#powerrail
      I_Contact( #DONE )
      { S7_Templates := "SrcType := WChar" } EQ_Contact(in1 := #UNICODE, in2 := WCHAR#'w')
      Move(in := 16#77, out1 => #ASCII_HEX)
      S_Coil( #DONE )
   END_RUNG
   RUNG wire#powerrail
      I_Contact( #DONE )
      { S7_Templates := "SrcType := WChar" } EQ_Contact(in1 := #UNICODE, in2 := WCHAR#'x')
      Move(in := 16#78, out1 => #ASCII_HEX)
      S_Coil( #DONE )
   END_RUNG
   RUNG wire#powerrail
      I_Contact( #DONE )
      { S7_Templates := "SrcType := WChar" } EQ_Contact(in1 := #UNICODE, in2 := WCHAR#'y')
      Move(in := 16#79, out1 => #ASCII_HEX)
      S_Coil( #DONE )
   END_RUNG
   RUNG wire#powerrail
      I_Contact( #DONE )
      { S7_Templates := "SrcType := WChar" } EQ_Contact(in1 := #UNICODE, in2 := WCHAR#'z')
      Move(in := 16#7A, out1 => #ASCII_HEX)
      S_Coil( #DONE )
   END_RUNG
   // the same network as SCL:
   IF NOT #DONE AND (#UNICODE = WCHAR#'u') THEN
       #ASCII_HEX := 16#75;
       #DONE := TRUE;
   END_IF;
   IF NOT #DONE AND (#UNICODE = WCHAR#'v') THEN
       #ASCII_HEX := 16#76;
       #DONE := TRUE;
   END_IF;
   IF NOT #DONE AND (#UNICODE = WCHAR#'w') THEN
       #ASCII_HEX := 16#77;
       #DONE := TRUE;
   END_IF;
   IF NOT #DONE AND (#UNICODE = WCHAR#'x') THEN
       #ASCII_HEX := 16#78;
       #DONE := TRUE;
   END_IF;
   IF NOT #DONE AND (#UNICODE = WCHAR#'y') THEN
       #ASCII_HEX := 16#79;
       #DONE := TRUE;
   END_IF;
   IF NOT #DONE AND (#UNICODE = WCHAR#'z') THEN
       #ASCII_HEX := 16#7A;
       #DONE := TRUE;
   END_IF;
END_REGION
END_FUNCTION

FUNCTION "Comm_FC" : Void
{ S7_Optimized_Access := 'TRUE' }
VERSION : 0.1
   VAR_TEMP 
      x : Int;
   END_VAR


BEGIN
	// Передача данных на шкафы скважин
	FOR #x := 1 TO 11 DO
	    "Comm_DB".SHUSKV[#x].Output.AI_LE_105_Result := "LE_105".Result;
	    "Comm_DB".SHUSKV[#x].Output.AI_LE_106_Result := "LE_106".Result;
	    "Comm_DB".SHUSKV[#x].Output.AI_LE_107_Result := "LE_107".Result;
	    "Comm_DB".SHUSKV[#x].Output.AI_LE_108_Result := "LE_108".Result;
	    "Comm_DB".SHUSKV[#x].Output.AI_TE_101_Result := "TE_101".Result;
	    "Comm_DB".SHUSKV[#x].Output.AI_TE_102_Result := "TE_102".Result;
	    "Comm_DB".SHUSKV[#x].Output.AI_TE_103_Result := "TE_103".Result;
	    "Comm_DB".SHUSKV[#x].Output.AI_TE_104_Result := "TE_104".Result;
	END_FOR;
	
	// Передача данных на скаду
	"Comm_Scada".Input.LE_105_Result := "LE_105".Result;
	"Comm_Scada".Input.LE_106_Result := "LE_106".Result;
	"Comm_Scada".Input.LE_107_Result := "LE_107".Result;
	"Comm_Scada".Input.LE_108_Result := "LE_108".Result;
	"Comm_Scada".Input.TE_101_Result := "TE_101".Result;
	"Comm_Scada".Input.TE_102_Result := "TE_102".Result;
	"Comm_Scada".Input.TE_103_Result := "TE_103".Result;
	"Comm_Scada".Input.TE_104_Result := "TE_104".Result;
	"Comm_Scada".Input.LE_105_Alarm := "LE_105".Alarms;
	"Comm_Scada".Input.LE_106_Alarm := "LE_106".Alarms;
	"Comm_Scada".Input.LE_107_Alarm := "LE_107".Alarms;
	"Comm_Scada".Input.LE_108_Alarm := "LE_108".Alarms;
	"Comm_Scada".Input.TE_101_Alarm := "TE_101".Alarms;
	"Comm_Scada".Input.TE_102_Alarm := "TE_102".Alarms;
	"Comm_Scada".Input.TE_103_Alarm := "TE_103".Alarms;
	"Comm_Scada".Input.TE_104_Alarm := "TE_104".Alarms;
	
	
END_FUNCTION

FUNCTION_BLOCK "Route_Control"
{ S7_Optimized_Access := 'TRUE' }
VERSION : 0.1

BEGIN
	//Общие компоненты - открыть
	IF "SKV_Logic_DB".Start THEN
	    "KP_REQ".KP_2_1[1] := TRUE;
	    "KP_REQ".KP_2_1[2] := TRUE;
	    "KP_REQ".KP_2_2[1] := TRUE;
	END_IF;
	
	//Общие компоненты - закрыть
	IF NOT "SKV_Logic_DB".Start
	    AND NOT ("Comm_SKV_1".From_SKV.Status = 1)
	    AND NOT ("Comm_SKV_2".From_SKV.Status = 1)
	    AND NOT ("Comm_SKV_3".From_SKV.Status = 1)
	    AND NOT ("Comm_SKV_13".From_SKV.Status = 1)
	    AND NOT ("Comm_SKV_14".From_SKV.Status = 1)
	    AND NOT ("Comm_SKV_15".From_SKV.Status = 1)
	    AND NOT ("Comm_SKV_20".From_SKV.Status = 1)
	    AND NOT ("Comm_SKV_21".From_SKV.Status = 1)
	    AND NOT ("Comm_SKV_22".From_SKV.Status = 1)
	    AND NOT ("Comm_SKV_23".From_SKV.Status = 1)
	THEN
	    "KP_REQ".KP_2_1[1] := FALSE;
	    "KP_REQ".KP_2_1[2] := FALSE;
	    "KP_REQ".KP_2_2[1] := FALSE;
	    "KP_REQ".KP_2_3[1] := FALSE;
	    "KP_REQ".KP_2_3[2] := FALSE;
	    "KP_REQ".KP_2_4[1] := FALSE;
	    "KP_REQ".KP_2_4[2] := FALSE;
	    "KP_REQ".KP_2_5[1] := FALSE;
	    "KP_REQ".KP_2_5[2] := FALSE;
	    "KP_REQ".KP_2_5[3] := FALSE;
	    "KP_REQ".KP_2_6[1] := FALSE;
	    "KP_REQ".KP_2_6[2] := FALSE;
	    "KP_REQ".KP_2_6[3] := FALSE;
	    "KP_REQ".KP_2_6[4] := FALSE;
	    "KP_REQ".KP_2_6[5] := FALSE;
	    "KP_REQ".KP_2_6[6] := FALSE;
	    "KP_REQ".KP_2_7[1] := FALSE;
	    "KP_REQ".KP_2_7[2] := FALSE;
	    "KP_REQ".KP_2_7[3] := FALSE;
	    "KP_REQ".KP_2_7[4] := FALSE;
	    "KP_REQ".KP_2_7[5] := FALSE;
	    "KP_REQ".KP_2_7[6] := FALSE;
	    "KP_REQ".KP_2_7[7] := FALSE;
	    "KP_REQ".KP_2_7[8] := FALSE;
	    "KP_REQ".KP_2_8[1] := FALSE;
	    "KP_REQ".KP_2_9[1] := FALSE;
	    "KP_REQ".KP_2_9[2] := FALSE;
	    "KP_REQ".KP_2_10[1] := FALSE;
	    "KP_REQ".KP_2_10[2] := FALSE;
	END_IF;
	    
	// СКВ-3 - Сборка маршрута
	IF "SKV_Logic_DB".Start AND "Comm_SKV_3".To_SKV.CMD.REQ THEN
	        "KP_REQ".KP_2_8[1] := TRUE;
	END_IF;
	//разборка маршрута
	IF NOT "SKV_Logic_DB".Start OR (NOT ("Comm_SKV_3".From_SKV.Status = 1) AND NOT "Comm_SKV_3".To_SKV.CMD.REQ) THEN
	    "KP_REQ".KP_2_8[1] := FALSE;
	END_IF;
	
	// СКВ-23 - Сборка маршрута
	IF "SKV_Logic_DB".Start AND "Comm_SKV_23".To_SKV.CMD.REQ THEN
	    "KP_REQ".KP_2_10[1] := TRUE;
	    "KP_REQ".KP_2_9[2] := TRUE;
	    "KP_REQ".KP_2_7[2] := TRUE;
	    "KP_REQ".KP_2_7[1] := TRUE;
	END_IF;
	//разборка маршрута
	IF NOT "SKV_Logic_DB".Start OR (NOT ("Comm_SKV_23".From_SKV.Status = 1) AND NOT "Comm_SKV_23".To_SKV.CMD.REQ) THEN
	    "KP_REQ".KP_2_10[1] := FALSE;
	END_IF;
	
	// СКВ-15 - Сборка маршрута
	IF "SKV_Logic_DB".Start AND "Comm_SKV_15".To_SKV.CMD.REQ THEN
	    "KP_REQ".KP_2_10[2] := TRUE;
	    "KP_REQ".KP_2_9[2] := TRUE;
	    "KP_REQ".KP_2_7[2] := TRUE;
	    "KP_REQ".KP_2_7[1] := TRUE;
	END_IF;
	//разборка маршрута
	IF NOT "SKV_Logic_DB".Start OR (NOT ("Comm_SKV_15".From_SKV.Status = 1) AND NOT "Comm_SKV_15".To_SKV.CMD.REQ) THEN
	    "KP_REQ".KP_2_10[2] := FALSE;
	END_IF;
	
	//Общий участок СКВ-23 и СКВ-15
	IF NOT "SKV_Logic_DB".Start OR ((NOT ("Comm_SKV_23".From_SKV.Status = 1) AND NOT "Comm_SKV_23".To_SKV.CMD.REQ)
	    AND (NOT ("Comm_SKV_15".From_SKV.Status = 1) AND NOT "Comm_SKV_15".To_SKV.CMD.REQ)) THEN
	    "KP_REQ".KP_2_9[2] := TRUE;
	END_IF;
	
	// СКВ-12 - Сборка маршрута
	IF "SKV_Logic_DB".Start AND "Comm_SKV_12".To_SKV.CMD.REQ THEN
	    "KP_REQ".KP_2_9[1] := TRUE;
	    "KP_REQ".KP_2_7[2] := TRUE;
	    "KP_REQ".KP_2_7[1] := TRUE;
	END_IF;
	//разборка маршрута
	IF NOT "SKV_Logic_DB".Start OR (NOT ("Comm_SKV_12".From_SKV.Status = 1) AND NOT "Comm_SKV_12".To_SKV.CMD.REQ) THEN
	    "KP_REQ".KP_2_9[1] := FALSE;
	END_IF;
	
	//Общий участок СКВ-23, СКВ-15 и СКВ-12
	IF NOT "SKV_Logic_DB".Start OR ((NOT ("Comm_SKV_23".From_SKV.Status = 1) AND NOT "Comm_SKV_23".To_SKV.CMD.REQ)
	    AND (NOT ("Comm_SKV_15".From_SKV.Status = 1) AND NOT "Comm_SKV_15".To_SKV.CMD.REQ)
	    AND (NOT ("Comm_SKV_12".From_SKV.Status = 1) AND NOT "Comm_SKV_12".To_SKV.CMD.REQ))
	THEN
	    "KP_REQ".KP_2_7[2] := FALSE;
	END_IF;
	
	
	// СКВ-13 - Сборка маршрута
	IF "SKV_Logic_DB".Start AND "Comm_SKV_23".To_SKV.CMD.REQ THEN
	    "KP_REQ".KP_2_7[6] := TRUE;
	    "KP_REQ".KP_2_7[3] := TRUE;
	    "KP_REQ".KP_2_7[4] := TRUE;
	    "KP_REQ".KP_2_7[5] := TRUE;
	    "KP_REQ".KP_2_7[1] := TRUE;
	END_IF;
	//разборка маршрута
	IF NOT "SKV_Logic_DB".Start OR (NOT ("Comm_SKV_13".From_SKV.Status = 1) AND NOT "Comm_SKV_13".To_SKV.CMD.REQ) THEN
	    "KP_REQ".KP_2_7[6] := FALSE;
	END_IF;
	
	// СКВ-14 - Сборка маршрута
	IF "SKV_Logic_DB".Start AND "Comm_SKV_14".To_SKV.CMD.REQ THEN
	    "KP_REQ".KP_2_6[1] := TRUE;
	    
	    "KP_REQ".KP_2_6[3] := TRUE;
	    
	    "KP_REQ".KP_2_7[8] := TRUE;
	    "KP_REQ".KP_2_7[3] := TRUE;
	    "KP_REQ".KP_2_7[4] := TRUE;
	    "KP_REQ".KP_2_7[5] := TRUE;
	END_IF;
	//разборка маршрута
	IF NOT "SKV_Logic_DB".Start OR (NOT ("Comm_SKV_14".From_SKV.Status = 1) AND NOT "Comm_SKV_14".To_SKV.CMD.REQ) THEN
	    "KP_REQ".KP_2_6[1] := FALSE;
	END_IF;
	
	// СКВ-1 - сборка маршрута
	IF "SKV_Logic_DB".Start AND "Comm_SKV_1".To_SKV.CMD.REQ THEN
	    "KP_REQ".KP_2_3[1] := TRUE;
	    "KP_REQ".KP_2_4[1] := TRUE;
	    "KP_REQ".KP_2_5[1] := TRUE;
	    
	    "KP_REQ".KP_2_6[2] := TRUE;
	    "KP_REQ".KP_2_6[3] := TRUE;
	    
	    "KP_REQ".KP_2_7[8] := TRUE;
	    "KP_REQ".KP_2_7[3] := TRUE;
	    "KP_REQ".KP_2_7[4] := TRUE;
	    "KP_REQ".KP_2_7[5] := TRUE;
	END_IF;
	//разборка маршрута
	IF NOT "SKV_Logic_DB".Start OR (NOT ("Comm_SKV_1".From_SKV.Status = 1) AND NOT "Comm_SKV_1".To_SKV.CMD.REQ) THEN
	    "KP_REQ".KP_2_3[1] := FALSE;
	END_IF;
	
	// СКВ-20 - сборка маршрута
	IF "SKV_Logic_DB".Start AND "Comm_SKV_20".To_SKV.CMD.REQ THEN
	    "KP_REQ".KP_2_3[2] := TRUE;
	    "KP_REQ".KP_2_4[1] := TRUE;
	    "KP_REQ".KP_2_5[1] := TRUE;
	    
	    "KP_REQ".KP_2_6[2] := TRUE;
	    "KP_REQ".KP_2_6[3] := TRUE;
	    
	    "KP_REQ".KP_2_7[8] := TRUE;
	    "KP_REQ".KP_2_7[3] := TRUE;
	    "KP_REQ".KP_2_7[4] := TRUE;
	    "KP_REQ".KP_2_7[5] := TRUE;
	END_IF;
	//разборка маршрута
	IF NOT "SKV_Logic_DB".Start OR (NOT ("Comm_SKV_20".From_SKV.Status = 1) AND NOT "Comm_SKV_20".To_SKV.CMD.REQ) THEN
	    "KP_REQ".KP_2_3[1] := FALSE;
	END_IF;
	
	//Общий участок
	IF NOT "SKV_Logic_DB".Start OR ((NOT ("Comm_SKV_1".From_SKV.Status = 1) AND NOT "Comm_SKV_1".To_SKV.CMD.REQ)
	    AND (NOT ("Comm_SKV_20".From_SKV.Status = 1) AND NOT "Comm_SKV_20".To_SKV.CMD.REQ))
	THEN
	    "KP_REQ".KP_2_4[1] := FALSE;
	END_IF;
	
	// СКВ-21 - сборка маршрута
	IF "SKV_Logic_DB".Start AND "Comm_SKV_21".To_SKV.CMD.REQ THEN
	    "KP_REQ".KP_2_4[2] := TRUE;
	    "KP_REQ".KP_2_5[1] := TRUE;
	    
	    "KP_REQ".KP_2_6[2] := TRUE;
	    "KP_REQ".KP_2_6[3] := TRUE;
	    
	    "KP_REQ".KP_2_7[8] := TRUE;
	    "KP_REQ".KP_2_7[3] := TRUE;
	    "KP_REQ".KP_2_7[4] := TRUE;
	    "KP_REQ".KP_2_7[5] := TRUE;
	END_IF;
	//разборка маршрута
	IF NOT "SKV_Logic_DB".Start OR (NOT ("Comm_SKV_21".From_SKV.Status = 1) AND NOT "Comm_SKV_21".To_SKV.CMD.REQ) THEN
	    "KP_REQ".KP_2_4[2] := FALSE;
	END_IF;
	
	//Общий участок
	IF NOT "SKV_Logic_DB".Start OR ((NOT ("Comm_SKV_1".From_SKV.Status = 1) AND NOT "Comm_SKV_1".To_SKV.CMD.REQ)
	    AND (NOT ("Comm_SKV_20".From_SKV.Status = 1) AND NOT "Comm_SKV_20".To_SKV.CMD.REQ)
	    AND (NOT ("Comm_SKV_21".From_SKV.Status = 1) AND NOT "Comm_SKV_21".To_SKV.CMD.REQ))
	THEN
	    "KP_REQ".KP_2_5[1] := FALSE;
	END_IF;
	
	
	// СКВ-22 - сборка маршрута
	IF "SKV_Logic_DB".Start AND "Comm_SKV_22".To_SKV.CMD.REQ THEN
	    "KP_REQ".KP_2_5[2] := TRUE;
	    
	    "KP_REQ".KP_2_6[2] := TRUE;
	    "KP_REQ".KP_2_6[3] := TRUE;
	    
	    "KP_REQ".KP_2_7[8] := TRUE;
	    "KP_REQ".KP_2_7[3] := TRUE;
	    "KP_REQ".KP_2_7[4] := TRUE;
	    "KP_REQ".KP_2_7[5] := TRUE;
	END_IF;
	//разборка маршрута
	IF NOT "SKV_Logic_DB".Start OR (NOT ("Comm_SKV_22".From_SKV.Status = 1) AND NOT "Comm_SKV_22".To_SKV.CMD.REQ) THEN
	    "KP_REQ".KP_2_5[3] := FALSE;
	END_IF;
	
END_FUNCTION_BLOCK

FUNCTION "SKV_Select" : Void
{ S7_Optimized_Access := 'TRUE' }
VERSION : 0.1
   VAR_INPUT 
      Limit : Int;   // Общее количество устр-ва
   END_VAR

   VAR_OUTPUT 
      Ready : Bool;   // Готовность выбранного устр-ва
      Status : Int;   // Статус выбранного устр--ва
   END_VAR

   VAR_IN_OUT 
      C : Real;   // Вес приоритета устр-ва
      REQ : Bool;   // Запрос обработки данных
      Mode : Bool;   // Команда - 0 - останов, 1 - запуск
      Number : Int;   // Номер устр-ва
   END_VAR

   VAR_TEMP 
      x : Int;
   END_VAR


BEGIN
	//контроль запроса на выбор насоса для запуска
	IF #REQ THEN
	    #C := 0.0;
	    #Number := 0;
	    #Status := -1;
	    #Ready := FALSE;
	    
	    FOR #x := 1 TO #Limit DO
	        //выбор максимального веса
	        IF "SKV_Main_DB".One[#x].C >= #C THEN
	            #C := "SKV_Main_DB".One[#x].C;
	        END_IF;
	    END_FOR;
	    
	    //проходим по всему списку насосов
	    FOR #x := 1 TO #Limit DO
	        //выбор насоса для запуска
	        IF #Mode THEN
	            //проверяем приоритетность запуска для остановленных насосов
	            IF "SKV_Main_DB".One[#x].C <= #C AND "SKV_Main_DB".One[#x].CMD.Ready AND NOT "SKV_Main_DB".One[#x].CMD.Start_M THEN
	                #C := "SKV_Main_DB".One[#x].C;           //сохраняем приоритет в буфер
	                #Number := #x;                           //возвращаем номер насоса для запуска
	                #Ready := "SKV_Main_DB".One[#x].CMD.Ready;
	                #Status := "SKV_Main_DB".One[#x].Status;
	            END_IF;
	        END_IF;
	    END_FOR;
	    
	    FOR #x := 1 TO #Limit DO
	        
	        //выбор максимального веса
	        IF "SKV_Main_DB".One[#x].C <= #C THEN
	            #C := "SKV_Main_DB".One[#x].C;
	        END_IF;
	        
	    END_FOR;
	    
	    //проходим по всему списку насосов
	    FOR #x := 1 TO #Limit DO
	        
	        //выбор насоса для останова
	        IF NOT #Mode THEN
	            //проверяем приоритетность запуска для остановки насосов
	            IF "SKV_Main_DB".One[#x].C >= #C AND "SKV_Main_DB".One[#x].Status = 3 AND "SKV_Main_DB".One[#x].CMD.Start_M THEN
	                #C := "SKV_Main_DB".One[#x].C;  //сохраняем приоритет в буфер
	                #Number := #x;                  //возвращаем номер насоса для запуска
	                #Ready := "SKV_Main_DB".One[#x].CMD.Ready;
	            END_IF;
	        END_IF;
	    END_FOR;
	    
	    //снятие флага запуска
	    #REQ := FALSE;
	END_IF;
	
	
	
	
	
END_FUNCTION

FUNCTION_BLOCK "SKV_cnt"
{ S7_Optimized_Access := 'FALSE' }
VERSION : 0.1
   VAR 
      CMD : Struct   // Команды и атрибуты
         Select : Bool;   // - выбрать устр-во
         Mode : Bool;   // - режим выбора (1 - пуск, 0 - останов)
         Rotation : Bool;   // - ротация устр-в
         Load : Bool;   // - ввод недостающего устр-ва
         Reload : Bool;   // - ввод резервного устр-ва
         Deload : Bool;   // - вывод устр-ва при аварии
         Add : Bool;   // - запрос ввода нового устр-ва
         REQ : Int;   // - количество требуемых устр-в
      END_STRUCT;
      Data : Struct   // Данные
         Ready : Bool;   // - готовность выбранного насоса
         Add_Ready : Bool;   // - система готова к вводу нового устр-ва
         C : Real;   // - вес проверяемого устр-ва
         REQ : Int;   // - кол-во запущенных устр-в
         N : Int;   // - номер выбранного устр-ва
         Status : Int;   // - статус выбранного устр-ва
         N_On : Int;   // - устр-во для запуска при ротации
         N_Off : Int;   // - устр-во для останова при ротации
      END_STRUCT;
      Step : Int;   // Шаг операции
      dev : Int;
      Clock : Array[0..4] of "Time_S";   // Блок таймеров
   END_VAR


BEGIN
	//Выбор насоса для запуска или останова
	"SKV_Select"(Limit:= "SKV_Main_DB".cnt.All,
	             Ready=>#Data.Ready,
	             Status=>#Data.Status,
	             C:=#Data.C,
	             REQ:=#CMD.Select,
	             Mode:=#CMD.Mode,
	             Number:=#Data.N);
	
	//Отключение
	IF #CMD.REQ = 0 AND "SKV_Main_DB".cnt.Work = 0 THEN
	    #Step := 0;
	    #Data.REQ := 0;
	END_IF;
	
	//Запуск первого устр-ва
	CASE #Step OF
	    0:  //появилась команда запуска
	        IF #CMD.REQ > 0 THEN
	            #CMD.Select := TRUE;
	            #CMD.Mode := TRUE;
	            #Step := 1;
	        END_IF;
	    1:  //выбор завершён
	        IF NOT #CMD.Select THEN
	            IF #Data.Ready THEN
	                #Step := 2;
	            ELSE
	                #Step := 3;
	            END_IF;
	        END_IF;
	    2:  //проверка выбора - устр-во готово
	        "SKV_Main_DB".One[#Data.N].CMD.Start_A := TRUE;
	        #Data.REQ := #Data.REQ + 1;
	        IF #Data.REQ >= #CMD.REQ THEN
	            #Step := 9;
	        ELSE
	            #Step := 0;
	        END_IF;
	    3:  //проверка выбора - устр-во не готово
	        IF "SKV_Main_DB".cnt.Ready >= #CMD.REQ THEN
	            IF #Data.REQ < #CMD.REQ THEN
	                #Step := 0;
	            END_IF;
	        ELSE
	            #CMD.REQ := #Data.REQ;
	            #Step := 9;
	        END_IF;
	    9:  //первое устр-во успешно запущено
	        IF "SKV_Main_DB".cnt.Work >= 1 THEN
	            #Step := 10;
	        END_IF;
	END_CASE;
	
	//Добавление устр-ва в работу
	CASE #Step OF
	    10: //проверка необходимости добавления нового устр-ва
	        IF (#CMD.REQ > #Data.REQ OR #CMD.Reload OR #CMD.Load) AND "SKV_Main_DB".cnt.Ready > 0 THEN
	            #CMD.Select := TRUE;
	            #CMD.Mode := TRUE;
	            #Step := 11;
	        END_IF;
	    11: //проверка выбора
	        IF NOT #CMD.Select THEN
	            IF #Data.Status = 0 THEN
	                #Step := 12;
	            ELSE
	                #Step := 10;
	            END_IF;
	        END_IF;
	    12: //запуск выбранного устр-ва
	        "SKV_Main_DB".One[#Data.N].CMD.Start_A := TRUE;
	        IF "SKV_Main_DB".One[#Data.N].Status = "SKV_Main_DB".One[#Data.N].Mode THEN
	            #CMD.Add := TRUE;
	            "SKV_Main_DB".One[#Data.N].SP.Auto := "SKV_Main_DB".SP.Point;
	            "SKV_Main_DB".One[#Data.N].Mode := 2;
	            #Step := #Step + 1;
	        END_IF;
	    13: //выход на режим ввода нового устр-ва
	        IF "SKV_Main_DB".One[#Data.N].Status = "SKV_Main_DB".One[#Data.N].Mode THEN
	            IF (NOT #CMD.Reload AND NOT #CMD.Load AND #Data.Add_Ready) OR (#CMD.Reload OR #CMD.Load) THEN
	                #CMD.Add := FALSE;
	                "SKV_Main_DB".One[#Data.N].Mode := 3;
	                #Step := #Step + 1;
	            END_IF;
	        END_IF;
	    14: //выход на штатный режим работы
	        IF NOT #CMD.Reload THEN
	            IF #Data.REQ < #CMD.REQ THEN
	                #Data.REQ := #Data.REQ + 1;
	            END_IF;
	        END_IF;
	        #Step := 19;
	    19: //пауза перед следующей операцией
	        #CMD.Reload := FALSE;
	        #CMD.Load := FALSE;
	        #CMD.Add := FALSE;
	        #Clock[0].Start := TRUE;
	        IF #Clock[0]."Exit" THEN
	            #Step := 10;
	        END_IF;
	END_CASE;
	
	//Вывод устр-ва из работы
	CASE #Step OF
	    10: //проверка необходимости добавления нового устр-ва
	        IF (#CMD.REQ < #Data.REQ OR #CMD.Deload) THEN
	            #CMD.Select := TRUE;
	            #CMD.Mode := FALSE;
	            #Step := 21;
	        END_IF;
	    21: //проверка выбора и снижение производительности устр-ва
	        IF NOT #CMD.Select THEN
	            "SKV_Main_DB".One[#Data.N].Mode := 5;
	            IF "SKV_Main_DB".One[#Data.N].Status = "SKV_Main_DB".One[#Data.N].Mode THEN
	                IF NOT #CMD.Deload THEN
	                    #Data.REQ := #Data.REQ - 1;
	                END_IF;
	                #Step := 22;
	            END_IF;
	        END_IF;
	    22: //отключение устр-ва
	        "SKV_Main_DB".One[#Data.N].Mode := 6;
	        #Step := 29;
	    29: //пауза перед следующей операцией
	        #CMD.Deload := FALSE;
	        #Clock[1].Start := TRUE;
	        IF #Clock[1]."Exit" THEN
	            #Step := 10;
	        END_IF;
	END_CASE;
	
	//Ротация
	CASE #Step OF
	    10: //проверка необходимости добавления нового устр-ва
	        IF #CMD.Rotation THEN
	            #CMD.Select := TRUE;
	            #CMD.Mode := TRUE;
	            #Step := 31;
	        END_IF;
	    31: //выбор устр-ва для запуска
	        IF NOT #CMD.Select THEN
	            #Data.N_On := #Data.N;
	            #Step := #Step + 1;
	        END_IF;
	    32: //выбор устр-ва для останова
	        #CMD.Select := TRUE;
	        #CMD.Mode := FALSE;
	        #Step := #Step + 1;
	    33: //выбор устр-ва для останова
	        IF NOT #CMD.Select THEN
	            #Data.N_Off := #Data.N;
	            #Step := #Step + 1;
	        END_IF;
	    34: //выключение нового устр-ва и замедление работающего
	        "SKV_Main_DB".One[#Data.N_On].CMD.Start_A := TRUE;
	        "SKV_Main_DB".One[#Data.N_On].Mode := 1;
	        IF "SKV_Main_DB".One[#Data.N_On].Status = "SKV_Main_DB".One[#Data.N_On].Mode THEN
	            "SKV_Main_DB".One[#Data.N_Off].Mode := 5;
	            IF "SKV_Main_DB".One[#Data.N_Off].Status = "SKV_Main_DB".One[#Data.N_Off].Mode THEN
	                #Step := #Step + 1;
	            END_IF;
	        END_IF;
	    35: //отключение и выравнивание производительности
	        "SKV_Main_DB".One[#Data.N_Off].Mode := 6;
	        #CMD.Add := TRUE;
	        "SKV_Main_DB".One[#Data.N_On].SP.Auto := "SKV_Main_DB".SP.Point;
	        "SKV_Main_DB".One[#Data.N_On].Mode := 2;
	        IF "SKV_Main_DB".One[#Data.N_On].Status = "SKV_Main_DB".One[#Data.N_On].Mode THEN
	            #Step := 39;
	        END_IF;
	    39: //пауза перед следующей операцией
	        #CMD.Reload := FALSE;
	        #Clock[2].Start := TRUE;
	        IF #Clock[2]."Exit" THEN
	            #Step := 10;
	        END_IF;
	END_CASE;
	
	//call timers
	FOR #dev := 0 TO 4 DO
	    #Clock[#dev]();
	END_FOR;
	            
	        
END_FUNCTION_BLOCK

DATA_BLOCK "Main_Logick_DB"   // DB1
VERSION : 0.1
// stored: AutoNumber true, DBAccessibleFromOPCUA true, DBAccessibleFromWebserver true, InstanceOfName Main_Logick, InstanceOfType FB
"Main_Logick"
BEGIN
   Time_Contrast_SKV.SP_D := 3;
   Time_Contrast_SKV.SP_H := 0;
   Time_Contrast_SKV.SP_M := 0;
   Time_Contrast_SKV.SP_S := 0;
END_DATA_BLOCK

DATA_BLOCK "PID_ex_DB"   // DB7
VERSION : 0.1
// stored: AutoNumber true, DBAccessibleFromOPCUA true, DBAccessibleFromWebserver true, InstanceOfName PID_ex, InstanceOfType FB
"PID_ex"
BEGIN
   pos[0..15] := FALSE;
END_DATA_BLOCK

DATA_BLOCK "Put_Get_DB"   // DB2
VERSION : 0.1
// stored: AutoNumber true, DBAccessibleFromOPCUA true, DBAccessibleFromWebserver true, InstanceOfName Put_Get, InstanceOfType FB
"Put_Get"
BEGIN
END_DATA_BLOCK

DATA_BLOCK "Comm_SKV_1"   // DB1001
VERSION : 0.1
// stored: AutoNumber false, DBAccessibleFromOPCUA true, DBAccessibleFromWebserver true, InstanceOfName Comm_SKV, InstanceOfType FB
"Comm_SKV"
BEGIN
END_DATA_BLOCK

DATA_BLOCK "Comm_SKV_12"   // DB1012
VERSION : 0.1
// stored: AutoNumber false, DBAccessibleFromOPCUA true, DBAccessibleFromWebserver true, InstanceOfName Comm_SKV, InstanceOfType FB
"Comm_SKV"
BEGIN
END_DATA_BLOCK

DATA_BLOCK "Comm_SKV_13"   // DB1013
VERSION : 0.1
// stored: AutoNumber false, DBAccessibleFromOPCUA true, DBAccessibleFromWebserver true, InstanceOfName Comm_SKV, InstanceOfType FB
"Comm_SKV"
BEGIN
END_DATA_BLOCK

DATA_BLOCK "Comm_SKV_14"   // DB1014
VERSION : 0.1
// stored: AutoNumber false, DBAccessibleFromOPCUA true, DBAccessibleFromWebserver true, InstanceOfName Comm_SKV, InstanceOfType FB
"Comm_SKV"
BEGIN
END_DATA_BLOCK

DATA_BLOCK "Comm_SKV_15"   // DB1015
VERSION : 0.1
// stored: AutoNumber false, DBAccessibleFromOPCUA true, DBAccessibleFromWebserver true, InstanceOfName Comm_SKV, InstanceOfType FB
"Comm_SKV"
BEGIN
END_DATA_BLOCK

DATA_BLOCK "Comm_SKV_2"   // DB1002
VERSION : 0.1
// stored: AutoNumber false, DBAccessibleFromOPCUA true, DBAccessibleFromWebserver true, InstanceOfName Comm_SKV, InstanceOfType FB
"Comm_SKV"
BEGIN
END_DATA_BLOCK

DATA_BLOCK "Comm_SKV_20"   // DB1020
VERSION : 0.1
// stored: AutoNumber false, DBAccessibleFromOPCUA true, DBAccessibleFromWebserver true, InstanceOfName Comm_SKV, InstanceOfType FB
"Comm_SKV"
BEGIN
END_DATA_BLOCK

DATA_BLOCK "Comm_SKV_21"   // DB1021
VERSION : 0.1
// stored: AutoNumber false, DBAccessibleFromOPCUA true, DBAccessibleFromWebserver true, InstanceOfName Comm_SKV, InstanceOfType FB
"Comm_SKV"
BEGIN
END_DATA_BLOCK

DATA_BLOCK "Comm_SKV_22"   // DB1022
VERSION : 0.1
// stored: AutoNumber false, DBAccessibleFromOPCUA true, DBAccessibleFromWebserver true, InstanceOfName Comm_SKV, InstanceOfType FB
"Comm_SKV"
BEGIN
END_DATA_BLOCK

DATA_BLOCK "Comm_SKV_23"   // DB1023
VERSION : 0.1
// stored: AutoNumber false, DBAccessibleFromOPCUA true, DBAccessibleFromWebserver true, InstanceOfName Comm_SKV, InstanceOfType FB
"Comm_SKV"
BEGIN
END_DATA_BLOCK

DATA_BLOCK "Comm_SKV_3"   // DB1003
VERSION : 0.1
// stored: AutoNumber false, DBAccessibleFromOPCUA true, DBAccessibleFromWebserver true, InstanceOfName Comm_SKV, InstanceOfType FB
"Comm_SKV"
BEGIN
END_DATA_BLOCK

DATA_BLOCK "Route_Check_DB"   // DB8
VERSION : 0.1
// stored: AutoNumber true, DBAccessibleFromOPCUA true, DBAccessibleFromWebserver true, InstanceOfName Route_Check, InstanceOfType FB
"Route_Check"
BEGIN
END_DATA_BLOCK

DATA_BLOCK "Route_Control_DB"   // DB13
VERSION : 0.1
// stored: AutoNumber true, DBAccessibleFromOPCUA true, DBAccessibleFromWebserver true, InstanceOfName Route_Control, InstanceOfType FB
"Route_Control"
BEGIN
END_DATA_BLOCK

DATA_BLOCK "SKV_Logic_DB"   // DB12
VERSION : 0.1
// stored: AutoNumber true, DBAccessibleFromOPCUA true, DBAccessibleFromWebserver true, InstanceOfName SKV_Logic, InstanceOfType FB
"SKV_Logic"
BEGIN
END_DATA_BLOCK

DATA_BLOCK "SKV_Main_DB"   // DB15
VERSION : 0.1
// stored: AutoNumber true, DBAccessibleFromOPCUA true, DBAccessibleFromWebserver true, InstanceOfName SKV_Main, InstanceOfType FB
"SKV_Main"
BEGIN
   One[0..11].SP_Use := TRUE;
   One[0].Mode := 0;
   One[1..11].Mode := 1;
   One[0..11].C := 0.0;
   One[0..11].SP.Low_Percent := 85.0;
   One[0..11].SP.Min := 30.0;
   One[0..11].SP.Max := 45.0;
   One[0..11].SP.Delta := 10.0;
END_DATA_BLOCK

DATA_BLOCK "SKV_cnt_DB"   // DB4
VERSION : 0.1
// stored: AutoNumber true, DBAccessibleFromOPCUA true, DBAccessibleFromWebserver true, InstanceOfName SKV_cnt, InstanceOfType FB
"SKV_cnt"
BEGIN
   Clock[0].SP := 10;
   Clock[1..4].SP := 2;
END_DATA_BLOCK

DATA_BLOCK "ModBus_DB"   // DB20
VERSION : 0.1
// stored: AutoNumber false, DBAccessibleFromOPCUA true, DBAccessibleFromWebserver true, InstanceOfName ModBus, InstanceOfType FB
"ModBus"
BEGIN
END_DATA_BLOCK

DATA_BLOCK "ModBus_TCP_DB"   // DB40
VERSION : 0.1
// stored: AutoNumber false, DBAccessibleFromOPCUA true, DBAccessibleFromWebserver true, InstanceOfName ModBus_TCP, InstanceOfType FB
"ModBus_TCP"
BEGIN
   CONNECT.InterfaceId := 64;
   CONNECT.ID := 1;
   CONNECT.ConnectionType := 11;
   CONNECT.RemoteAddress.ADDR[1] := 192;
   CONNECT.RemoteAddress.ADDR[2] := 168;
   CONNECT.RemoteAddress.ADDR[3] := 0;
   CONNECT.RemoteAddress.ADDR[4] := 10;
   CONNECT.RemotePort := 502;
END_DATA_BLOCK

DATA_BLOCK "AIx_DB"   // DB220
VERSION : 0.1
// stored: AutoNumber false, DBAccessibleFromOPCUA true, DBAccessibleFromWebserver true, InstanceOfName AIx, InstanceOfType FB
"AIx"
BEGIN
END_DATA_BLOCK

DATA_BLOCK "AOx_DB"   // DB230
VERSION : 0.1
// stored: AutoNumber false, DBAccessibleFromOPCUA true, DBAccessibleFromWebserver true, InstanceOfName AOx, InstanceOfType FB
"AOx"
BEGIN
END_DATA_BLOCK

DATA_BLOCK "DIx_1_DB"   // DB200
VERSION : 0.1
// stored: AutoNumber false, DBAccessibleFromOPCUA true, DBAccessibleFromWebserver true, InstanceOfName DIx_1, InstanceOfType FB
"DIx_1"
BEGIN
   AllBlock.Use.Inverse := FALSE;
   AllBlock.Use.Indirect := TRUE;
   AllBlock.ADDR_Byte := 0;
   AllBlock.ADDR_Bit := 0;
   AllBlock.Filter_On.SP := 16#02;
   AllBlock.Filter_Off.SP := 16#02;
   RM_impulse.Use.Inverse := FALSE;
   RM_impulse.Use.Indirect := TRUE;
   RM_impulse.ADDR_Byte := 0;
   RM_impulse.ADDR_Bit := 1;
   RM_impulse.Filter_On.SP := 16#02;
   RM_impulse.Filter_Off.SP := 16#02;
   "3Fok".Use.Inverse := FALSE;
   "3Fok".Use.Indirect := TRUE;
   "3Fok".ADDR_Byte := 0;
   "3Fok".ADDR_Bit := 2;
   "3Fok".Filter_On.SP := 16#02;
   "3Fok".Filter_Off.SP := 16#02;
   signal_4.Use.Inverse := FALSE;
   signal_4.Use.Indirect := TRUE;
   signal_4.ADDR_Byte := 0;
   signal_4.ADDR_Bit := 9;
   signal_4.Filter_On.SP := 16#02;
   signal_4.Filter_Off.SP := 16#02;
   signal_5.Use.Inverse := FALSE;
   signal_5.Use.Indirect := TRUE;
   signal_5.ADDR_Byte := 0;
   signal_5.ADDR_Bit := 9;
   signal_5.Filter_On.SP := 16#02;
   signal_5.Filter_Off.SP := 16#02;
   signal_6.Use.Inverse := FALSE;
   signal_6.Use.Indirect := TRUE;
   signal_6.ADDR_Byte := 0;
   signal_6.ADDR_Bit := 9;
   signal_6.Filter_On.SP := 16#02;
   signal_6.Filter_Off.SP := 16#02;
   signal_7.Use.Inverse := FALSE;
   signal_7.Use.Indirect := TRUE;
   signal_7.ADDR_Byte := 0;
   signal_7.ADDR_Bit := 9;
   signal_7.Filter_On.SP := 16#02;
   signal_7.Filter_Off.SP := 16#02;
   signal_8.Use.Inverse := FALSE;
   signal_8.Use.Indirect := TRUE;
   signal_8.ADDR_Byte := 0;
   signal_8.ADDR_Bit := 9;
   signal_8.Filter_On.SP := 16#02;
   signal_8.Filter_Off.SP := 16#02;
   signal_9.Use.Inverse := FALSE;
   signal_9.Use.Indirect := TRUE;
   signal_9.ADDR_Byte := 0;
   signal_9.ADDR_Bit := 9;
   signal_9.Filter_On.SP := 16#02;
   signal_9.Filter_Off.SP := 16#02;
   signal_10.Use.Inverse := FALSE;
   signal_10.Use.Indirect := TRUE;
   signal_10.ADDR_Byte := 0;
   signal_10.ADDR_Bit := 9;
   signal_10.Filter_On.SP := 16#02;
   signal_10.Filter_Off.SP := 16#02;
   signal_11.Use.Inverse := FALSE;
   signal_11.Use.Indirect := TRUE;
   signal_11.ADDR_Byte := 0;
   signal_11.ADDR_Bit := 9;
   signal_11.Filter_On.SP := 16#02;
   signal_11.Filter_Off.SP := 16#02;
   signal_12.Use.Inverse := FALSE;
   signal_12.Use.Indirect := TRUE;
   signal_12.ADDR_Byte := 0;
   signal_12.ADDR_Bit := 9;
   signal_12.Filter_On.SP := 16#02;
   signal_12.Filter_Off.SP := 16#02;
END_DATA_BLOCK

DATA_BLOCK "DOx_1_DB"   // DB210
VERSION : 0.1
// stored: AutoNumber false, DBAccessibleFromOPCUA true, DBAccessibleFromWebserver true, InstanceOfName DOx_1, InstanceOfType FB
"DOx_1"
BEGIN
   All_Alarm.Use.Inverse := FALSE;
   All_Alarm.Use.Indirect := TRUE;
   All_Alarm.Use.Impulse := FALSE;
   All_Alarm.ADDR_Byte := 0;
   All_Alarm.ADDR_Bit := 1;
   All_Alarm.T_Impulse.SP := 16#02;
   command_2.Use.Inverse := FALSE;
   command_2.Use.Indirect := TRUE;
   command_2.Use.Impulse := FALSE;
   command_2.ADDR_Byte := 0;
   command_2.ADDR_Bit := 9;
   command_2.T_Impulse.SP := 16#02;
   command_3.Use.Inverse := FALSE;
   command_3.Use.Indirect := TRUE;
   command_3.Use.Impulse := FALSE;
   command_3.ADDR_Byte := 0;
   command_3.ADDR_Bit := 9;
   command_3.T_Impulse.SP := 16#02;
   command_4.Use.Inverse := FALSE;
   command_4.Use.Indirect := TRUE;
   command_4.Use.Impulse := FALSE;
   command_4.ADDR_Byte := 0;
   command_4.ADDR_Bit := 9;
   command_4.T_Impulse.SP := 16#02;
   command_5.Use.Inverse := FALSE;
   command_5.Use.Indirect := TRUE;
   command_5.Use.Impulse := FALSE;
   command_5.ADDR_Byte := 0;
   command_5.ADDR_Bit := 9;
   command_5.T_Impulse.SP := 16#02;
   command_6.Use.Inverse := FALSE;
   command_6.Use.Indirect := TRUE;
   command_6.Use.Impulse := FALSE;
   command_6.ADDR_Byte := 0;
   command_6.ADDR_Bit := 9;
   command_6.T_Impulse.SP := 16#02;
   command_7.Use.Inverse := FALSE;
   command_7.Use.Indirect := TRUE;
   command_7.Use.Impulse := FALSE;
   command_7.ADDR_Byte := 0;
   command_7.ADDR_Bit := 9;
   command_7.T_Impulse.SP := 16#02;
   command_8.Use.Inverse := FALSE;
   command_8.Use.Indirect := TRUE;
   command_8.Use.Impulse := FALSE;
   command_8.ADDR_Byte := 0;
   command_8.ADDR_Bit := 9;
   command_8.T_Impulse.SP := 16#02;
   command_9.Use.Inverse := FALSE;
   command_9.Use.Indirect := TRUE;
   command_9.Use.Impulse := FALSE;
   command_9.ADDR_Byte := 0;
   command_9.ADDR_Bit := 9;
   command_9.T_Impulse.SP := 16#02;
   command_10.Use.Inverse := FALSE;
   command_10.Use.Indirect := TRUE;
   command_10.Use.Impulse := FALSE;
   command_10.ADDR_Byte := 0;
   command_10.ADDR_Bit := 9;
   command_10.T_Impulse.SP := 16#02;
   command_11.Use.Inverse := FALSE;
   command_11.Use.Indirect := TRUE;
   command_11.Use.Impulse := FALSE;
   command_11.ADDR_Byte := 0;
   command_11.ADDR_Bit := 9;
   command_11.T_Impulse.SP := 16#02;
   command_12.Use.Inverse := FALSE;
   command_12.Use.Indirect := TRUE;
   command_12.Use.Impulse := FALSE;
   command_12.ADDR_Byte := 0;
   command_12.ADDR_Bit := 9;
   command_12.T_Impulse.SP := 16#02;
END_DATA_BLOCK

DATA_BLOCK "Motors_DB"   // DB240
VERSION : 0.1
// stored: AutoNumber false, DBAccessibleFromOPCUA true, DBAccessibleFromWebserver true, InstanceOfName Motors, InstanceOfType FB
"Motors"
BEGIN
END_DATA_BLOCK

DATA_BLOCK "PIDx_DB"   // DB260
VERSION : 0.1
// stored: AutoNumber false, DBAccessibleFromOPCUA true, DBAccessibleFromWebserver true, InstanceOfName PIDx, InstanceOfType FB
"PIDx"
BEGIN
END_DATA_BLOCK

DATA_BLOCK "Valves_DB"   // DB250
VERSION : 0.1
// stored: AutoNumber false, DBAccessibleFromOPCUA true, DBAccessibleFromWebserver true, InstanceOfName Valves, InstanceOfType FB
"Valves"
BEGIN
END_DATA_BLOCK

DATA_BLOCK "KP_1_DB"   // DB521
VERSION : 0.1
// stored: AutoNumber false, DBAccessibleFromOPCUA true, DBAccessibleFromWebserver true, InstanceOfName KP_1, InstanceOfType FB
"KP_1"
BEGIN
   KP[0..10].Use.QF := FALSE;
   KP[0..10].Use.KM_Open := FALSE;
   KP[0..10].Use.KM_Close := FALSE;
   KP[0..10].Use.Open := TRUE;
   KP[0..10].Use.Close := TRUE;
   KP[0..10].Use.One_KM := FALSE;
   KP[0..10].Use.Air := FALSE;
   KP[0..10].Use.Cross := FALSE;
   KP[0..10].Use.CMD_Open := TRUE;
   KP[0..10].Use.CMD_Close := FALSE;
   KP[0..10].Use.Local_Keys := FALSE;
   KP[0..10].Use.CWF := FALSE;
   KP[0].Clock[0].SP := 10;
   KP[0].Clock[1..4].SP := 2;
   KP[1].Clock[0].SP := 10;
   KP[1].Clock[1..4].SP := 2;
   KP[2].Clock[0].SP := 10;
   KP[2].Clock[1..4].SP := 2;
   KP[3].Clock[0].SP := 10;
   KP[3].Clock[1..4].SP := 2;
   KP[4].Clock[0].SP := 10;
   KP[4].Clock[1..4].SP := 2;
   KP[5].Clock[0].SP := 10;
   KP[5].Clock[1..4].SP := 2;
   KP[6].Clock[0].SP := 10;
   KP[6].Clock[1..4].SP := 2;
   KP[7].Clock[0].SP := 10;
   KP[7].Clock[1..4].SP := 2;
   KP[8].Clock[0].SP := 10;
   KP[8].Clock[1..4].SP := 2;
   KP[9].Clock[0].SP := 10;
   KP[9].Clock[1..4].SP := 2;
   KP[10].Clock[0].SP := 10;
   KP[10].Clock[1..4].SP := 2;
   KP[0].CodeID := 0;
   KP[1].CodeID := 1;
   KP[2].CodeID := 2;
   KP[3].CodeID := 3;
   KP[4].CodeID := 4;
   KP[5].CodeID := 5;
   KP[6..10].CodeID := 0;
   KP[0..10].Speed := 16#00;
END_DATA_BLOCK

DATA_BLOCK "KP_2_10_DB"   // DB520
VERSION : 0.1
// stored: AutoNumber false, DBAccessibleFromOPCUA true, DBAccessibleFromWebserver true, InstanceOfName KP_2_10, InstanceOfType FB
"KP_2_10"
BEGIN
   KP[0..10].Use.QF := FALSE;
   KP[0..10].Use.KM_Open := FALSE;
   KP[0..10].Use.KM_Close := FALSE;
   KP[0..10].Use.Open := TRUE;
   KP[0..10].Use.Close := TRUE;
   KP[0..10].Use.One_KM := FALSE;
   KP[0..10].Use.Air := FALSE;
   KP[0..10].Use.Cross := FALSE;
   KP[0..10].Use.CMD_Open := TRUE;
   KP[0..10].Use.CMD_Close := FALSE;
   KP[0..10].Use.Local_Keys := FALSE;
   KP[0..10].Use.CWF := FALSE;
   KP[0].Clock[0].SP := 10;
   KP[0].Clock[1..4].SP := 2;
   KP[1].Clock[0].SP := 10;
   KP[1].Clock[1..2].SP := 2;
   KP[1].Clock[3..4].SP := 99;
   KP[2].Clock[0].SP := 10;
   KP[2].Clock[1..2].SP := 2;
   KP[2].Clock[3..4].SP := 99;
   KP[3].Clock[0].SP := 10;
   KP[3].Clock[1..4].SP := 2;
   KP[4].Clock[0].SP := 10;
   KP[4].Clock[1..4].SP := 2;
   KP[5].Clock[0].SP := 10;
   KP[5].Clock[1..4].SP := 2;
   KP[6].Clock[0].SP := 10;
   KP[6].Clock[1..4].SP := 2;
   KP[7].Clock[0].SP := 10;
   KP[7].Clock[1..4].SP := 2;
   KP[8].Clock[0].SP := 10;
   KP[8].Clock[1..4].SP := 2;
   KP[9].Clock[0].SP := 10;
   KP[9].Clock[1..4].SP := 2;
   KP[10].Clock[0].SP := 10;
   KP[10].Clock[1..4].SP := 2;
   KP[0].CodeID := 0;
   KP[1].CodeID := 1;
   KP[2].CodeID := 2;
   KP[3..10].CodeID := 0;
   KP[0..10].Speed := 16#00;
END_DATA_BLOCK

DATA_BLOCK "KP_2_1_DB"   // DB511
VERSION : 0.1
// stored: AutoNumber false, DBAccessibleFromOPCUA true, DBAccessibleFromWebserver true, InstanceOfName KP_2_1, InstanceOfType FB
"KP_2_1"
BEGIN
   KP[0..10].Use.QF := FALSE;
   KP[0..10].Use.KM_Open := FALSE;
   KP[0..10].Use.KM_Close := FALSE;
   KP[0..10].Use.Open := TRUE;
   KP[0..10].Use.Close := TRUE;
   KP[0..10].Use.One_KM := FALSE;
   KP[0..10].Use.Air := FALSE;
   KP[0..10].Use.Cross := FALSE;
   KP[0..10].Use.CMD_Open := TRUE;
   KP[0..10].Use.CMD_Close := FALSE;
   KP[0..10].Use.Local_Keys := FALSE;
   KP[0..10].Use.CWF := FALSE;
   KP[0].Clock[0].SP := 10;
   KP[0].Clock[1..4].SP := 2;
   KP[1].Clock[0].SP := 10;
   KP[1].Clock[1..2].SP := 2;
   KP[1].Clock[3..4].SP := 99;
   KP[2].Clock[0].SP := 10;
   KP[2].Clock[1..2].SP := 2;
   KP[2].Clock[3..4].SP := 99;
   KP[3].Clock[0].SP := 10;
   KP[3].Clock[1..2].SP := 2;
   KP[3].Clock[3..4].SP := 99;
   KP[4].Clock[0].SP := 10;
   KP[4].Clock[1..4].SP := 2;
   KP[5].Clock[0].SP := 10;
   KP[5].Clock[1..4].SP := 2;
   KP[6].Clock[0].SP := 10;
   KP[6].Clock[1..4].SP := 2;
   KP[7].Clock[0].SP := 10;
   KP[7].Clock[1..4].SP := 2;
   KP[8].Clock[0].SP := 10;
   KP[8].Clock[1..4].SP := 2;
   KP[9].Clock[0].SP := 10;
   KP[9].Clock[1..4].SP := 2;
   KP[10].Clock[0].SP := 10;
   KP[10].Clock[1..4].SP := 2;
   KP[0].CodeID := 0;
   KP[1].CodeID := 1;
   KP[2].CodeID := 2;
   KP[3].CodeID := 3;
   KP[4..10].CodeID := 0;
   KP[0..10].Speed := 16#00;
END_DATA_BLOCK

DATA_BLOCK "KP_2_2_DB"   // DB512
VERSION : 0.1
// stored: AutoNumber false, DBAccessibleFromOPCUA true, DBAccessibleFromWebserver true, InstanceOfName KP_2_2, InstanceOfType FB
"KP_2_2"
BEGIN
   KP[0..10].Use.QF := FALSE;
   KP[0..10].Use.KM_Open := FALSE;
   KP[0..10].Use.KM_Close := FALSE;
   KP[0..10].Use.Open := TRUE;
   KP[0..10].Use.Close := TRUE;
   KP[0..10].Use.One_KM := FALSE;
   KP[0..10].Use.Air := FALSE;
   KP[0..10].Use.Cross := FALSE;
   KP[0..10].Use.CMD_Open := TRUE;
   KP[0..10].Use.CMD_Close := FALSE;
   KP[0..10].Use.Local_Keys := FALSE;
   KP[0..10].Use.CWF := FALSE;
   KP[0].Clock[0].SP := 10;
   KP[0].Clock[1..4].SP := 2;
   KP[1].Clock[0].SP := 10;
   KP[1].Clock[1..2].SP := 2;
   KP[1].Clock[3..4].SP := 99;
   KP[2].Clock[0].SP := 10;
   KP[2].Clock[1..4].SP := 2;
   KP[3].Clock[0].SP := 10;
   KP[3].Clock[1..4].SP := 2;
   KP[4].Clock[0].SP := 10;
   KP[4].Clock[1..4].SP := 2;
   KP[5].Clock[0].SP := 10;
   KP[5].Clock[1..4].SP := 2;
   KP[6].Clock[0].SP := 10;
   KP[6].Clock[1..4].SP := 2;
   KP[7].Clock[0].SP := 10;
   KP[7].Clock[1..4].SP := 2;
   KP[8].Clock[0].SP := 10;
   KP[8].Clock[1..4].SP := 2;
   KP[9].Clock[0].SP := 10;
   KP[9].Clock[1..4].SP := 2;
   KP[10].Clock[0].SP := 10;
   KP[10].Clock[1..4].SP := 2;
   KP[0].CodeID := 0;
   KP[1].CodeID := 1;
   KP[2..10].CodeID := 0;
   KP[0..10].Speed := 16#00;
END_DATA_BLOCK

DATA_BLOCK "KP_2_3_DB"   // DB513
VERSION : 0.1
// stored: AutoNumber false, DBAccessibleFromOPCUA true, DBAccessibleFromWebserver true, InstanceOfName KP_2_3, InstanceOfType FB
"KP_2_3"
BEGIN
   KP[0..10].Use.QF := FALSE;
   KP[0..10].Use.KM_Open := FALSE;
   KP[0..10].Use.KM_Close := FALSE;
   KP[0..10].Use.Open := TRUE;
   KP[0..10].Use.Close := TRUE;
   KP[0..10].Use.One_KM := FALSE;
   KP[0..10].Use.Air := FALSE;
   KP[0..10].Use.Cross := FALSE;
   KP[0..10].Use.CMD_Open := TRUE;
   KP[0..10].Use.CMD_Close := FALSE;
   KP[0..10].Use.Local_Keys := FALSE;
   KP[0..10].Use.CWF := FALSE;
   KP[0].Clock[0].SP := 10;
   KP[0].Clock[1..4].SP := 2;
   KP[1].Clock[0].SP := 10;
   KP[1].Clock[1..2].SP := 2;
   KP[1].Clock[3..4].SP := 99;
   KP[2].Clock[0].SP := 10;
   KP[2].Clock[1..2].SP := 2;
   KP[2].Clock[3..4].SP := 99;
   KP[3].Clock[0].SP := 10;
   KP[3].Clock[1..4].SP := 2;
   KP[4].Clock[0].SP := 10;
   KP[4].Clock[1..4].SP := 2;
   KP[5].Clock[0].SP := 10;
   KP[5].Clock[1..4].SP := 2;
   KP[6].Clock[0].SP := 10;
   KP[6].Clock[1..4].SP := 2;
   KP[7].Clock[0].SP := 10;
   KP[7].Clock[1..4].SP := 2;
   KP[8].Clock[0].SP := 10;
   KP[8].Clock[1..4].SP := 2;
   KP[9].Clock[0].SP := 10;
   KP[9].Clock[1..4].SP := 2;
   KP[10].Clock[0].SP := 10;
   KP[10].Clock[1..4].SP := 2;
   KP[0].CodeID := 0;
   KP[1].CodeID := 1;
   KP[2].CodeID := 2;
   KP[3..10].CodeID := 0;
   KP[0..10].Speed := 16#00;
END_DATA_BLOCK

DATA_BLOCK "KP_2_4_DB"   // DB514
VERSION : 0.1
// stored: AutoNumber false, DBAccessibleFromOPCUA true, DBAccessibleFromWebserver true, InstanceOfName KP_2_4, InstanceOfType FB
"KP_2_4"
BEGIN
   KP[0..10].Use.QF := FALSE;
   KP[0..10].Use.KM_Open := FALSE;
   KP[0..10].Use.KM_Close := FALSE;
   KP[0..10].Use.Open := TRUE;
   KP[0..10].Use.Close := TRUE;
   KP[0..10].Use.One_KM := FALSE;
   KP[0..10].Use.Air := FALSE;
   KP[0..10].Use.Cross := FALSE;
   KP[0..10].Use.CMD_Open := TRUE;
   KP[0..10].Use.CMD_Close := FALSE;
   KP[0..10].Use.Local_Keys := FALSE;
   KP[0..10].Use.CWF := FALSE;
   KP[0].Clock[0].SP := 10;
   KP[0].Clock[1..4].SP := 2;
   KP[1].Clock[0].SP := 10;
   KP[1].Clock[1..2].SP := 2;
   KP[1].Clock[3..4].SP := 99;
   KP[2].Clock[0].SP := 10;
   KP[2].Clock[1..2].SP := 2;
   KP[2].Clock[3].SP := 999;
   KP[2].Clock[4].SP := 99;
   KP[3].Clock[0].SP := 10;
   KP[3].Clock[1..4].SP := 2;
   KP[4].Clock[0].SP := 10;
   KP[4].Clock[1..4].SP := 2;
   KP[5].Clock[0].SP := 10;
   KP[5].Clock[1..4].SP := 2;
   KP[6].Clock[0].SP := 10;
   KP[6].Clock[1..4].SP := 2;
   KP[7].Clock[0].SP := 10;
   KP[7].Clock[1..4].SP := 2;
   KP[8].Clock[0].SP := 10;
   KP[8].Clock[1..4].SP := 2;
   KP[9].Clock[0].SP := 10;
   KP[9].Clock[1..4].SP := 2;
   KP[10].Clock[0].SP := 10;
   KP[10].Clock[1..4].SP := 2;
   KP[0].CodeID := 0;
   KP[1].CodeID := 2;
   KP[2].CodeID := 1;
   KP[3..10].CodeID := 0;
   KP[0..10].Speed := 16#00;
END_DATA_BLOCK

DATA_BLOCK "KP_2_5_DB"   // DB515
VERSION : 0.1
// stored: AutoNumber false, DBAccessibleFromOPCUA true, DBAccessibleFromWebserver true, InstanceOfName KP_2_5, InstanceOfType FB
"KP_2_5"
BEGIN
   KP[0..10].Use.QF := FALSE;
   KP[0..10].Use.KM_Open := FALSE;
   KP[0..10].Use.KM_Close := FALSE;
   KP[0..10].Use.Open := TRUE;
   KP[0..10].Use.Close := TRUE;
   KP[0..10].Use.One_KM := FALSE;
   KP[0..10].Use.Air := FALSE;
   KP[0..10].Use.Cross := FALSE;
   KP[0..10].Use.CMD_Open := TRUE;
   KP[0..10].Use.CMD_Close := FALSE;
   KP[0..10].Use.Local_Keys := FALSE;
   KP[0..10].Use.CWF := FALSE;
   KP[0].Clock[0].SP := 10;
   KP[0].Clock[1..4].SP := 2;
   KP[1].Clock[0].SP := 10;
   KP[1].Clock[1..2].SP := 2;
   KP[1].Clock[3..4].SP := 99;
   KP[2].Clock[0].SP := 10;
   KP[2].Clock[1..2].SP := 2;
   KP[2].Clock[3..4].SP := 99;
   KP[3].Clock[0].SP := 10;
   KP[3].Clock[1..2].SP := 2;
   KP[3].Clock[3..4].SP := 99;
   KP[4].Clock[0].SP := 10;
   KP[4].Clock[1..4].SP := 2;
   KP[5].Clock[0].SP := 10;
   KP[5].Clock[1..4].SP := 2;
   KP[6].Clock[0].SP := 10;
   KP[6].Clock[1..4].SP := 2;
   KP[7].Clock[0].SP := 10;
   KP[7].Clock[1..4].SP := 2;
   KP[8].Clock[0].SP := 10;
   KP[8].Clock[1..4].SP := 2;
   KP[9].Clock[0].SP := 10;
   KP[9].Clock[1..4].SP := 2;
   KP[10].Clock[0].SP := 10;
   KP[10].Clock[1..4].SP := 2;
   KP[0].CodeID := 0;
   KP[1].CodeID := 1;
   KP[2].CodeID := 2;
   KP[3].CodeID := 3;
   KP[4].CodeID := 2;
   KP[5].CodeID := 4;
   KP[6..10].CodeID := 0;
   KP[0..10].Speed := 16#00;
END_DATA_BLOCK

DATA_BLOCK "KP_2_6_DB"   // DB516
VERSION : 0.1
// stored: AutoNumber false, DBAccessibleFromOPCUA true, DBAccessibleFromWebserver true, InstanceOfName KP_2_6, InstanceOfType FB
"KP_2_6"
BEGIN
   KP[0..10].Use.QF := FALSE;
   KP[0..10].Use.KM_Open := FALSE;
   KP[0..10].Use.KM_Close := FALSE;
   KP[0..10].Use.Open := TRUE;
   KP[0..10].Use.Close := TRUE;
   KP[0..10].Use.One_KM := FALSE;
   KP[0..10].Use.Air := FALSE;
   KP[0..10].Use.Cross := FALSE;
   KP[0..10].Use.CMD_Open := TRUE;
   KP[0..10].Use.CMD_Close := FALSE;
   KP[0..10].Use.Local_Keys := FALSE;
   KP[0..10].Use.CWF := FALSE;
   KP[0].Clock[0].SP := 10;
   KP[0].Clock[1..2].SP := 2;
   KP[0].Clock[3..4].SP := 99;
   KP[1].Clock[0].SP := 10;
   KP[1].Clock[1..2].SP := 2;
   KP[1].Clock[3..4].SP := 99;
   KP[2].Clock[0].SP := 10;
   KP[2].Clock[1..2].SP := 2;
   KP[2].Clock[3..4].SP := 99;
   KP[3].Clock[0].SP := 10;
   KP[3].Clock[1..2].SP := 2;
   KP[3].Clock[3..4].SP := 99;
   KP[4].Clock[0].SP := 10;
   KP[4].Clock[1..2].SP := 2;
   KP[4].Clock[3..4].SP := 99;
   KP[5].Clock[0].SP := 10;
   KP[5].Clock[1..2].SP := 2;
   KP[5].Clock[3..4].SP := 99;
   KP[6].Clock[0].SP := 10;
   KP[6].Clock[1..2].SP := 2;
   KP[6].Clock[3..4].SP := 99;
   KP[7].Clock[0].SP := 10;
   KP[7].Clock[1..4].SP := 2;
   KP[8].Clock[0].SP := 10;
   KP[8].Clock[1..4].SP := 2;
   KP[9].Clock[0].SP := 10;
   KP[9].Clock[1..4].SP := 2;
   KP[10].Clock[0].SP := 10;
   KP[10].Clock[1..4].SP := 2;
   KP[0..1].CodeID := 1;
   KP[2].CodeID := 2;
   KP[3].CodeID := 3;
   KP[4].CodeID := 4;
   KP[5].CodeID := 6;
   KP[6].CodeID := 5;
   KP[7..10].CodeID := 0;
   KP[0..10].Speed := 16#00;
END_DATA_BLOCK

DATA_BLOCK "KP_2_7_DB"   // DB517
VERSION : 0.1
// stored: AutoNumber false, DBAccessibleFromOPCUA true, DBAccessibleFromWebserver true, InstanceOfName KP_2_7, InstanceOfType FB
"KP_2_7"
BEGIN
   KP[0..10].Use.QF := FALSE;
   KP[0..10].Use.KM_Open := FALSE;
   KP[0..10].Use.KM_Close := FALSE;
   KP[0..10].Use.Open := TRUE;
   KP[0..10].Use.Close := TRUE;
   KP[0..10].Use.One_KM := FALSE;
   KP[0..10].Use.Air := FALSE;
   KP[0..10].Use.Cross := FALSE;
   KP[0..10].Use.CMD_Open := TRUE;
   KP[0..10].Use.CMD_Close := FALSE;
   KP[0..10].Use.Local_Keys := FALSE;
   KP[0..10].Use.CWF := FALSE;
   KP[0].Clock[0].SP := 10;
   KP[0].Clock[1..4].SP := 2;
   KP[1].Clock[0].SP := 10;
   KP[1].Clock[1..2].SP := 2;
   KP[1].Clock[3..4].SP := 99;
   KP[2].Clock[0].SP := 10;
   KP[2].Clock[1..2].SP := 2;
   KP[2].Clock[3..4].SP := 99;
   KP[3].Clock[0].SP := 10;
   KP[3].Clock[1..2].SP := 2;
   KP[3].Clock[3..4].SP := 99;
   KP[4].Clock[0].SP := 10;
   KP[4].Clock[1..2].SP := 2;
   KP[4].Clock[3..4].SP := 99;
   KP[5].Clock[0].SP := 10;
   KP[5].Clock[1..2].SP := 2;
   KP[5].Clock[3..4].SP := 99;
   KP[6].Clock[0].SP := 10;
   KP[6].Clock[1..2].SP := 2;
   KP[6].Clock[3..4].SP := 99;
   KP[7].Clock[0].SP := 10;
   KP[7].Clock[1..2].SP := 2;
   KP[7].Clock[3..4].SP := 99;
   KP[8].Clock[0].SP := 10;
   KP[8].Clock[1..2].SP := 2;
   KP[8].Clock[3..4].SP := 99;
   KP[9].Clock[0].SP := 10;
   KP[9].Clock[1..4].SP := 2;
   KP[10].Clock[0].SP := 10;
   KP[10].Clock[1..4].SP := 2;
   KP[0].CodeID := 0;
   KP[1].CodeID := 2;
   KP[2].CodeID := 1;
   KP[3].CodeID := 8;
   KP[4].CodeID := 5;
   KP[5].CodeID := 3;
   KP[6].CodeID := 7;
   KP[7].CodeID := 4;
   KP[8].CodeID := 6;
   KP[9..10].CodeID := 0;
   KP[0..10].Speed := 16#00;
END_DATA_BLOCK

DATA_BLOCK "KP_2_8_DB"   // DB518
VERSION : 0.1
// stored: AutoNumber false, DBAccessibleFromOPCUA true, DBAccessibleFromWebserver true, InstanceOfName KP_2_8, InstanceOfType FB
"KP_2_8"
BEGIN
   KP[0..10].Use.QF := FALSE;
   KP[0..10].Use.KM_Open := FALSE;
   KP[0..10].Use.KM_Close := FALSE;
   KP[0..10].Use.Open := TRUE;
   KP[0..10].Use.Close := TRUE;
   KP[0..10].Use.One_KM := FALSE;
   KP[0..10].Use.Air := FALSE;
   KP[0..10].Use.Cross := FALSE;
   KP[0..10].Use.CMD_Open := TRUE;
   KP[0..10].Use.CMD_Close := FALSE;
   KP[0..10].Use.Local_Keys := FALSE;
   KP[0..10].Use.CWF := FALSE;
   KP[0].Clock[0].SP := 10;
   KP[0].Clock[1..4].SP := 2;
   KP[1].Clock[0].SP := 10;
   KP[1].Clock[1..2].SP := 2;
   KP[1].Clock[3..4].SP := 99;
   KP[2].Clock[0].SP := 10;
   KP[2].Clock[1..4].SP := 2;
   KP[3].Clock[0].SP := 10;
   KP[3].Clock[1..4].SP := 2;
   KP[4].Clock[0].SP := 10;
   KP[4].Clock[1..4].SP := 2;
   KP[5].Clock[0].SP := 10;
   KP[5].Clock[1..4].SP := 2;
   KP[6].Clock[0].SP := 10;
   KP[6].Clock[1..4].SP := 2;
   KP[7].Clock[0].SP := 10;
   KP[7].Clock[1..4].SP := 2;
   KP[8].Clock[0].SP := 10;
   KP[8].Clock[1..4].SP := 2;
   KP[9].Clock[0].SP := 10;
   KP[9].Clock[1..4].SP := 2;
   KP[10].Clock[0].SP := 10;
   KP[10].Clock[1..4].SP := 2;
   KP[0].CodeID := 0;
   KP[1].CodeID := 1;
   KP[2..10].CodeID := 0;
   KP[0..10].Speed := 16#00;
END_DATA_BLOCK

DATA_BLOCK "KP_2_9_DB"   // DB519
VERSION : 0.1
// stored: AutoNumber false, DBAccessibleFromOPCUA true, DBAccessibleFromWebserver true, InstanceOfName KP_2_9, InstanceOfType FB
"KP_2_9"
BEGIN
   KP[0..10].Use.QF := FALSE;
   KP[0..10].Use.KM_Open := FALSE;
   KP[0..10].Use.KM_Close := FALSE;
   KP[0..10].Use.Open := TRUE;
   KP[0..10].Use.Close := TRUE;
   KP[0..10].Use.One_KM := FALSE;
   KP[0..10].Use.Air := FALSE;
   KP[0..10].Use.Cross := FALSE;
   KP[0..10].Use.CMD_Open := TRUE;
   KP[0..10].Use.CMD_Close := FALSE;
   KP[0..10].Use.Local_Keys := FALSE;
   KP[0..10].Use.CWF := FALSE;
   KP[0].Clock[0].SP := 10;
   KP[0].Clock[1..4].SP := 2;
   KP[1].Clock[0].SP := 10;
   KP[1].Clock[1..2].SP := 2;
   KP[1].Clock[3..4].SP := 99;
   KP[2].Clock[0].SP := 10;
   KP[2].Clock[1..2].SP := 2;
   KP[2].Clock[3..4].SP := 99;
   KP[3].Clock[0].SP := 10;
   KP[3].Clock[1..4].SP := 2;
   KP[4].Clock[0].SP := 10;
   KP[4].Clock[1..4].SP := 2;
   KP[5].Clock[0].SP := 10;
   KP[5].Clock[1..4].SP := 2;
   KP[6].Clock[0].SP := 10;
   KP[6].Clock[1..4].SP := 2;
   KP[7].Clock[0].SP := 10;
   KP[7].Clock[1..4].SP := 2;
   KP[8].Clock[0].SP := 10;
   KP[8].Clock[1..4].SP := 2;
   KP[9].Clock[0].SP := 10;
   KP[9].Clock[1..4].SP := 2;
   KP[10].Clock[0].SP := 10;
   KP[10].Clock[1..4].SP := 2;
   KP[0].CodeID := 0;
   KP[1].CodeID := 2;
   KP[2].CodeID := 1;
   KP[3..10].CodeID := 0;
   KP[0..10].Speed := 16#00;
END_DATA_BLOCK

DATA_BLOCK "KP_2_DB"   // DB522
VERSION : 0.1
// stored: AutoNumber false, DBAccessibleFromOPCUA true, DBAccessibleFromWebserver true, InstanceOfName KP_2, InstanceOfType FB
"KP_2"
BEGIN
END_DATA_BLOCK

DATA_BLOCK "KP_3_DB"   // DB523
VERSION : 0.1
// stored: AutoNumber false, DBAccessibleFromOPCUA true, DBAccessibleFromWebserver true, InstanceOfName KP_3, InstanceOfType FB
"KP_3"
BEGIN
END_DATA_BLOCK

DATA_BLOCK "KP_4_DB"   // DB524
VERSION : 0.1
// stored: AutoNumber false, DBAccessibleFromOPCUA true, DBAccessibleFromWebserver true, InstanceOfName KP_4, InstanceOfType FB
"KP_4"
BEGIN
END_DATA_BLOCK

DATA_BLOCK "KP_5_DB"   // DB525
VERSION : 0.1
// stored: AutoNumber false, DBAccessibleFromOPCUA true, DBAccessibleFromWebserver true, InstanceOfName KP_5, InstanceOfType FB
"KP_5"
BEGIN
END_DATA_BLOCK

DATA_BLOCK "FB_DRV_Start_DB"   // DB100
VERSION : 0.1
// stored: AutoNumber false, DBAccessibleFromOPCUA true, DBAccessibleFromWebserver true, InstanceOfName FB_DRV_Start, InstanceOfType FB
"FB_DRV_Start"
BEGIN
END_DATA_BLOCK

DATA_BLOCK "Historian_DB"   // DB88
VERSION : 0.1
// stored: AutoNumber false, DBAccessibleFromOPCUA true, DBAccessibleFromWebserver true, InstanceOfName Historian, InstanceOfType FB
"Historian"
BEGIN
END_DATA_BLOCK

DATA_BLOCK "Time_SYS_DB"   // DB95
VERSION : 0.1
// stored: AutoNumber false, DBAccessibleFromOPCUA true, DBAccessibleFromWebserver true, InstanceOfName Time_SYS, InstanceOfType FB
"Time_SYS"
BEGIN
   TimeZone.Bias := 180;
   TimeZone.DaylightBias := 60;
   TimeZone.DaylightStartMonth := 3;
   TimeZone.DaylightStartWeek := 5;
   TimeZone.DaylightStartWeekday := 7;
   TimeZone.DaylightStartHour := 2;
   TimeZone.DaylightStartMinute := 0;
   TimeZone.StandardStartMonth := 10;
   TimeZone.StandardStartWeek := 5;
   TimeZone.StandardStartWeekday := 1;
   TimeZone.StandardStartHour := 3;
   TimeZone.StandardStartMinute := 0;
   TimeZone.TimeZoneName := 'GMT+3';
   SET_TIMEZONE.REQ := FALSE;
   SET_TIMEZONE.TimeZone.Bias := 180;
   SET_TIMEZONE.TimeZone.DaylightBias := 60;
   SET_TIMEZONE.TimeZone.DaylightStartMonth := 3;
   SET_TIMEZONE.TimeZone.DaylightStartWeek := 5;
   SET_TIMEZONE.TimeZone.DaylightStartWeekday := 7;
   SET_TIMEZONE.TimeZone.DaylightStartHour := 2;
   SET_TIMEZONE.TimeZone.DaylightStartMinute := 0;
   SET_TIMEZONE.TimeZone.StandardStartMonth := 10;
   SET_TIMEZONE.TimeZone.StandardStartWeek := 5;
   SET_TIMEZONE.TimeZone.StandardStartWeekday := 1;
   SET_TIMEZONE.TimeZone.StandardStartHour := 3;
   SET_TIMEZONE.TimeZone.StandardStartMinute := 0;
   SET_TIMEZONE.TimeZone.TimeZoneName := 'GMT+3';
   SET_TIMEZONE.DONE := FALSE;
   SET_TIMEZONE.BUSY := FALSE;
   SET_TIMEZONE.ERROR := FALSE;
   SET_TIMEZONE.STATUS := 16#7000;
   SET_TIMEZONE.LastScanREQ := FALSE;
END_DATA_BLOCK

DATA_BLOCK "LE_105"   // DB300
VERSION : 0.1
// stored: AutoNumber false, DBAccessibleFromOPCUA true, DBAccessibleFromWebserver true, InstanceOfName AI_ex, InstanceOfType FB
"AI_ex"
BEGIN
   Converter.Use_Min_In := FALSE;
   Converter.Use_Max_In := FALSE;
   Converter.Use_Min_Out := FALSE;
   Converter.Use_Max_Out := FALSE;
   Converter.IO := FALSE;
   Converter.Inverse := FALSE;
   Converter.Min_In := 0.0;
   Converter.Min_Out := 0.0;
   Converter.Max_In := 27700.0;
   Converter.Max_Out := 3.0;
   Tx[0..1].SP := 3.0;
   Tx[2..5].SP := 1.0;
   Tx[0..5].One := 0.1;
END_DATA_BLOCK

DATA_BLOCK "LE_106"   // DB301
VERSION : 0.1
// stored: AutoNumber false, DBAccessibleFromOPCUA true, DBAccessibleFromWebserver true, InstanceOfName AI_ex, InstanceOfType FB
"AI_ex"
BEGIN
   Converter.Use_Min_In := FALSE;
   Converter.Use_Max_In := FALSE;
   Converter.Use_Min_Out := FALSE;
   Converter.Use_Max_Out := FALSE;
   Converter.IO := FALSE;
   Converter.Inverse := FALSE;
   Converter.Min_In := 0.0;
   Converter.Min_Out := 0.0;
   Converter.Max_In := 27648.0;
   Converter.Max_Out := 3.0;
   Tx[0..1].SP := 3.0;
   Tx[2..5].SP := 1.0;
   Tx[0..5].One := 0.1;
END_DATA_BLOCK

DATA_BLOCK "LE_107"   // DB302
VERSION : 0.1
// stored: AutoNumber false, DBAccessibleFromOPCUA true, DBAccessibleFromWebserver true, InstanceOfName AI_ex, InstanceOfType FB
"AI_ex"
BEGIN
   Converter.Use_Min_In := FALSE;
   Converter.Use_Max_In := FALSE;
   Converter.Use_Min_Out := FALSE;
   Converter.Use_Max_Out := FALSE;
   Converter.IO := FALSE;
   Converter.Inverse := FALSE;
   Converter.Min_In := 0.0;
   Converter.Min_Out := 0.0;
   Converter.Max_In := 27648.0;
   Converter.Max_Out := 3.0;
   Tx[0..1].SP := 3.0;
   Tx[2..5].SP := 1.0;
   Tx[0..5].One := 0.1;
END_DATA_BLOCK

DATA_BLOCK "LE_108"   // DB303
VERSION : 0.1
// stored: AutoNumber false, DBAccessibleFromOPCUA true, DBAccessibleFromWebserver true, InstanceOfName AI_ex, InstanceOfType FB
"AI_ex"
BEGIN
   Converter.Use_Min_In := FALSE;
   Converter.Use_Max_In := FALSE;
   Converter.Use_Min_Out := FALSE;
   Converter.Use_Max_Out := FALSE;
   Converter.IO := FALSE;
   Converter.Inverse := FALSE;
   Converter.Min_In := 0.0;
   Converter.Min_Out := 0.0;
   Converter.Max_In := 27648.0;
   Converter.Max_Out := 3.0;
   Tx[0..1].SP := 3.0;
   Tx[2..5].SP := 1.0;
   Tx[0..5].One := 0.1;
END_DATA_BLOCK

DATA_BLOCK "LE_Final_DB"   // DB308
VERSION : 0.1
// stored: AutoNumber false, DBAccessibleFromOPCUA true, DBAccessibleFromWebserver true, InstanceOfName AI_ex, InstanceOfType FB
"AI_ex"
BEGIN
END_DATA_BLOCK

DATA_BLOCK "TE_101"   // DB304
VERSION : 0.1
// stored: AutoNumber false, DBAccessibleFromOPCUA true, DBAccessibleFromWebserver true, InstanceOfName AI_ex, InstanceOfType FB
"AI_ex"
BEGIN
   Converter.Use_Min_In := FALSE;
   Converter.Use_Max_In := FALSE;
   Converter.Use_Min_Out := FALSE;
   Converter.Use_Max_Out := FALSE;
   Converter.IO := FALSE;
   Converter.Inverse := FALSE;
   Converter.Min_In := 0.0;
   Converter.Min_Out := -10.0;
   Converter.Max_In := 27648.0;
   Converter.Max_Out := 60.0;
   Tx[0..1].SP := 3.0;
   Tx[2..5].SP := 1.0;
   Tx[0..5].One := 0.1;
END_DATA_BLOCK

DATA_BLOCK "TE_102"   // DB305
VERSION : 0.1
// stored: AutoNumber false, DBAccessibleFromOPCUA true, DBAccessibleFromWebserver true, InstanceOfName AI_ex, InstanceOfType FB
"AI_ex"
BEGIN
   Converter.Use_Min_In := FALSE;
   Converter.Use_Max_In := FALSE;
   Converter.Use_Min_Out := FALSE;
   Converter.Use_Max_Out := FALSE;
   Converter.IO := FALSE;
   Converter.Inverse := FALSE;
   Converter.Min_In := 0.0;
   Converter.Min_Out := -10.0;
   Converter.Max_In := 27648.0;
   Converter.Max_Out := 60.0;
   Tx[0..1].SP := 3.0;
   Tx[2..5].SP := 1.0;
   Tx[0..5].One := 0.1;
END_DATA_BLOCK

DATA_BLOCK "TE_103"   // DB306
VERSION : 0.1
// stored: AutoNumber false, DBAccessibleFromOPCUA true, DBAccessibleFromWebserver true, InstanceOfName AI_ex, InstanceOfType FB
"AI_ex"
BEGIN
   Converter.Use_Min_In := FALSE;
   Converter.Use_Max_In := FALSE;
   Converter.Use_Min_Out := FALSE;
   Converter.Use_Max_Out := FALSE;
   Converter.IO := FALSE;
   Converter.Inverse := FALSE;
   Converter.Min_In := 0.0;
   Converter.Min_Out := -10.0;
   Converter.Max_In := 27648.0;
   Converter.Max_Out := 60.0;
   Tx[0..1].SP := 3.0;
   Tx[2..5].SP := 1.0;
   Tx[0..5].One := 0.1;
END_DATA_BLOCK

DATA_BLOCK "TE_104"   // DB307
VERSION : 0.1
// stored: AutoNumber false, DBAccessibleFromOPCUA true, DBAccessibleFromWebserver true, InstanceOfName AI_ex, InstanceOfType FB
"AI_ex"
BEGIN
   Converter.Use_Min_In := FALSE;
   Converter.Use_Max_In := FALSE;
   Converter.Use_Min_Out := FALSE;
   Converter.Use_Max_Out := FALSE;
   Converter.IO := FALSE;
   Converter.Inverse := FALSE;
   Converter.Min_In := 0.0;
   Converter.Min_Out := -10.0;
   Converter.Max_In := 27648.0;
   Converter.Max_Out := 60.0;
   Tx[0..1].SP := 3.0;
   Tx[2..5].SP := 1.0;
   Tx[0..5].One := 0.1;
END_DATA_BLOCK

DATA_BLOCK "AO_example_DB"   // DB400
VERSION : 0.1
// stored: AutoNumber false, DBAccessibleFromOPCUA true, DBAccessibleFromWebserver true, InstanceOfName AO_ex, InstanceOfType FB
"AO_ex"
BEGIN
   Converter.Use_Min_In := FALSE;
   Converter.Use_Max_In := FALSE;
   Converter.Use_Min_Out := FALSE;
   Converter.Use_Max_Out := FALSE;
   Converter.IO := FALSE;
   Converter.Inverse := FALSE;
   Converter.Min_In := 0.0;
   Converter.Min_Out := 0.0;
   Converter.Max_In := 0.0;
   Converter.Max_Out := 0.0;
   Slow.Use_Up := FALSE;
   Slow.Use_Down := FALSE;
   Slow.Step_Up := 0.125;
   Slow.Step_Down := 0.125;
   Slow.T_Up.SP := 1.0;
   Slow.T_Up.One := 0.1;
   Slow.T_Down.SP := 1.0;
   Slow.T_Down.One := 0.1;
END_DATA_BLOCK

DATA_BLOCK "M_DA_example_DB"   // DB600
VERSION : 0.1
// stored: AutoNumber false, DBAccessibleFromOPCUA true, DBAccessibleFromWebserver true, InstanceOfName DRV_M_DA, InstanceOfType FB
"DRV_M_DA"
BEGIN
   Tx[0..3].SP := 2;
   Converter.Use_Min_In := FALSE;
   Converter.Use_Max_In := FALSE;
   Converter.Use_Min_Out := FALSE;
   Converter.Use_Max_Out := FALSE;
   Converter.IO := FALSE;
   Converter.Inverse := FALSE;
   Converter.Min_In := 0.0;
   Converter.Min_Out := 0.0;
   Converter.Max_In := 0.0;
   Converter.Max_Out := 0.0;
   Slow.Use_Up := FALSE;
   Slow.Use_Down := FALSE;
   Slow.Step_Up := 0.125;
   Slow.Step_Down := 0.125;
   Slow.T_Up.SP := 1.0;
   Slow.T_Up.One := 0.1;
   Slow.T_Down.SP := 1.0;
   Slow.T_Down.One := 0.1;
END_DATA_BLOCK

DATA_BLOCK "M_D_example_DB"   // DB500
VERSION : 0.1
// stored: AutoNumber false, DBAccessibleFromOPCUA true, DBAccessibleFromWebserver true, InstanceOfName DRV_M_D, InstanceOfType FB
"DRV_M_D"
BEGIN
   Tx[0..3].SP := 2;
END_DATA_BLOCK

DATA_BLOCK "PID_example_DB"   // DB900
VERSION : 0.1
// stored: AutoNumber false, DBAccessibleFromOPCUA true, DBAccessibleFromWebserver true, InstanceOfName PID_ex, InstanceOfType FB
"PID_ex"
BEGIN
   CMD.Vector := FALSE;
   pos[0..15] := FALSE;
END_DATA_BLOCK

DATA_BLOCK "DB_Reset_All"   // DB1099
{ S7_Optimized_Access := 'TRUE' }
// stored: AutoNumber true, DBAccessibleFromOPCUA true, DBAccessibleFromWebserver true, InstanceOfName IEC_TIMER, OfSystemLibElement IEC_TIMER, OfSystemLibVersion 1.0
"IEC_TIMER"
   // VAR
   //    PT : Time;
   //    ET { ExternalWritable := 'False'} : Time;
   //    IN : Bool;
   //    Q { ExternalWritable := 'False'} : Bool;
   // END_VAR
BEGIN
END_DATA_BLOCK

DATA_BLOCK "DB_pulse_01s"   // DB1100
{ S7_Optimized_Access := 'TRUE' }
// stored: AutoNumber true, DBAccessibleFromOPCUA true, DBAccessibleFromWebserver true, InstanceOfName IEC_TIMER, OfSystemLibElement IEC_TIMER, OfSystemLibVersion 1.0
"IEC_TIMER"
   // VAR
   //    PT : Time;
   //    ET { ExternalWritable := 'False'} : Time;
   //    IN : Bool;
   //    Q { ExternalWritable := 'False'} : Bool;
   // END_VAR
BEGIN
END_DATA_BLOCK

DATA_BLOCK "DB_pulse_05s"   // DB1101
{ S7_Optimized_Access := 'TRUE' }
// stored: AutoNumber true, DBAccessibleFromOPCUA true, DBAccessibleFromWebserver true, InstanceOfName IEC_TIMER, OfSystemLibElement IEC_TIMER, OfSystemLibVersion 1.0
"IEC_TIMER"
   // VAR
   //    PT : Time;
   //    ET { ExternalWritable := 'False'} : Time;
   //    IN : Bool;
   //    Q { ExternalWritable := 'False'} : Bool;
   // END_VAR
BEGIN
END_DATA_BLOCK

DATA_BLOCK "DB_pulse_10s"   // DB1104
{ S7_Optimized_Access := 'TRUE' }
// stored: AutoNumber true, DBAccessibleFromOPCUA true, DBAccessibleFromWebserver true, InstanceOfName IEC_TIMER, OfSystemLibElement IEC_TIMER, OfSystemLibVersion 1.0
"IEC_TIMER"
   // VAR
   //    PT : Time;
   //    ET { ExternalWritable := 'False'} : Time;
   //    IN : Bool;
   //    Q { ExternalWritable := 'False'} : Bool;
   // END_VAR
BEGIN
END_DATA_BLOCK

DATA_BLOCK "DB_pulse_1m"   // DB1106
{ S7_Optimized_Access := 'TRUE' }
// stored: AutoNumber true, DBAccessibleFromOPCUA true, DBAccessibleFromWebserver true, InstanceOfName IEC_TIMER, OfSystemLibElement IEC_TIMER, OfSystemLibVersion 1.0
"IEC_TIMER"
   // VAR
   //    PT : Time;
   //    ET { ExternalWritable := 'False'} : Time;
   //    IN : Bool;
   //    Q { ExternalWritable := 'False'} : Bool;
   // END_VAR
BEGIN
END_DATA_BLOCK

DATA_BLOCK "DB_pulse_1s"   // DB1102
{ S7_Optimized_Access := 'TRUE' }
// stored: AutoNumber true, DBAccessibleFromOPCUA true, DBAccessibleFromWebserver true, InstanceOfName IEC_TIMER, OfSystemLibElement IEC_TIMER, OfSystemLibVersion 1.0
"IEC_TIMER"
   // VAR
   //    PT : Time;
   //    ET { ExternalWritable := 'False'} : Time;
   //    IN : Bool;
   //    Q { ExternalWritable := 'False'} : Bool;
   // END_VAR
BEGIN
END_DATA_BLOCK

DATA_BLOCK "DB_pulse_30s"   // DB1105
{ S7_Optimized_Access := 'TRUE' }
// stored: AutoNumber true, DBAccessibleFromOPCUA true, DBAccessibleFromWebserver true, InstanceOfName IEC_TIMER, OfSystemLibElement IEC_TIMER, OfSystemLibVersion 1.0
"IEC_TIMER"
   // VAR
   //    PT : Time;
   //    ET { ExternalWritable := 'False'} : Time;
   //    IN : Bool;
   //    Q { ExternalWritable := 'False'} : Bool;
   // END_VAR
BEGIN
END_DATA_BLOCK

DATA_BLOCK "DB_pulse_5s"   // DB1103
{ S7_Optimized_Access := 'TRUE' }
// stored: AutoNumber true, DBAccessibleFromOPCUA true, DBAccessibleFromWebserver true, InstanceOfName IEC_TIMER, OfSystemLibElement IEC_TIMER, OfSystemLibVersion 1.0
"IEC_TIMER"
   // VAR
   //    PT : Time;
   //    ET { ExternalWritable := 'False'} : Time;
   //    IN : Bool;
   //    Q { ExternalWritable := 'False'} : Bool;
   // END_VAR
BEGIN
END_DATA_BLOCK

